(* IEC 61131-3 sources: Yaha/Documentation/Infomaterial/OSCAT/pcworx_building_100/pcworx_building_100/pcworx_building_100_module_export, 58 files *)

(* ---- building.IEC ---- *)
(*@PROPERTIES_EX@
TYPE: DATA_TYPE
LOCALE: 0
*)
(* ------------------------------------------- *)

TYPE oscat_TIMER_EVENT_DATA :
  STRUCT
	TYP          : BYTE;
	CHANNEL      : BYTE;
	DAY          : BYTE;
	START        : UDINT;
	DURATION     : TIME;
	LAND         : BYTE;
	LOR          : BYTE;
	LAST         : UDINT;
  END_STRUCT;
END_TYPE

TYPE
  oscat_TIMER_EVENT           : ARRAY [0..63]    OF oscat_TIMER_EVENT_DATA;
END_TYPE

(* ------------------------------------------- *)

TYPE
  oscat_T_AVG24         	  : ARRAY [0..47]   OF INT;

  oscat_TP4_qn                : ARRAY [0..3]    OF BOOL;

  oscat_bsa_X                 : ARRAY [0..2]    OF BYTE;
  oscat_blind_scene_array     : ARRAY [0..15]   OF oscat_bsa_X;

END_TYPE

(* ---- ACTUATOR_2P.ST ---- *)
(*@PROPERTIES_EX@
TYPE: POU
LOCALE: 0
IEC_LANGUAGE: ST
PLC_TYPE: independent
PROC_TYPE: independent
GROUP: ACTUATORS
*)
(*@KEY@:DESCRIPTION*)
version 2.1	24. jan. 2009
programmer 	hugo
tested by	oscat

this is an intelligent actuator interface for any 2point actuator like coil drive.
the 2Point actuator can only switch on/off and therefore the input must be converted to on/off cycles.
the interface can be programmed with double click on the symbol.
in addition a self_act_time and self_act_cycles ca be programmed to switch n times on/off every self_act_time to avoid a valve to freeze.
the input value must be between 0 and 255. with the setup variable sens one can specify what must be the minimum input to turn the valve on at all.
at the same time an input > 255-sens will turn the valve on at all times.
(*@KEY@:END_DESCRIPTION*)
FUNCTION_BLOCK ACTUATOR_2P

(*Group:Default*)

VAR_INPUT
	IN :	BYTE;
	TEST :	BOOL;
	ARE :	BOOL := TRUE;
	CYCLE_TIME :	TIME;
	SENS :	BYTE;
	SELF_ACT_TIME :	TIME;
	SELF_ACT_PULSE :	TIME;
	SELF_ACT_CYCLES :	INT := 1;
END_VAR

VAR_OUTPUT
	OUT :	BOOL;
	ARO :	BOOL;
END_VAR

VAR_IN_OUT
	ARX :	BOOL;
END_VAR

VAR
	timer :	AUTORUN;
	pwgen :	GEN_PULSE;
END_VAR

(*@KEY@: WORKSHEET
NAME: ACTUATOR_2P
IEC_LANGUAGE: ST
*)
(* run the autorun timer *)
timer(trun := MUL_T_AI(SELF_ACT_PULSE,2 * SELF_ACT_CYCLES), toff := SELF_ACT_TIME, Test := TEST, ARE := ARE, arx := ARX);
ARX := timer.ARX;
ARO := timer.ARO;

(* run the pulse width generator *)
IF aro THEN
	pwgen(PTL := SELF_ACT_PULSE, PTH := SELF_ACT_PULSE);
	out := pwgen.Q;
ELSIF in < sens THEN
	out := FALSE;
ELSIF BYTE_TO_USINT(in) > USINT#255 - BYTE_TO_USINT(sens) THEN
	out := TRUE;
ELSE
	pwgen.PTH := (CYCLE_TIME * BYTE_TO_TIME(BAND_B(IN,SENS))  ) / BYTE_TO_TIME(BYTE#255);
	pwgen.PTL := CYCLE_TIME - pwgen.PTH;
	pwgen();
	out := pwgen.Q;
END_IF;

(* revision history
hm	7.10.2006 		rev 1.1
	changed error pos could not reach 1 or 0 under certain conditions due to error in code.
	changed on and off in force and force_in for better usability.

hm	17.1.2007		rev 1.2
	deleted unused variable time_overflow

hm	15.9.2007		rev 1.3
	replaced time() with T_PLC_MS for compatibility and performance reasons

hm	19. 11 2007		rev 1.4
	replaced left over statement time() with tx

hm	27. 12. 2007	REV 1.5
	CHANGED CODE FOR BETTER PERFORMANCE

hm	21. oct. 2008	rev 1.6
	code optimized

hm	23. nov. 2008	rev 2.0
	new code using library modules

hm	24. jan. 2009	rev 2.1
	deleted unused var inb
*)
(*@KEY@: END_WORKSHEET *)
END_FUNCTION_BLOCK

(* ---- ACTUATOR_3P.ST ---- *)
(*@PROPERTIES_EX@
TYPE: POU
LOCALE: 0
IEC_LANGUAGE: ST
PLC_TYPE: independent
PROC_TYPE: independent
GROUP: ACTUATORS
*)
(*@KEY@:DESCRIPTION*)
version 2.0	28. jan 2010
programmer 	hugo
tested by		oscat

actuator_3P is an interface for a 3 point actuator.
a 3P actuator is a motor with 2 directions that drives a valve or flap. the position of the valve or flap is controlled by runtime of the motor foreward or backward.
the available inputs are:
IN specifies the position of the actuator, 0 = 0% and 255 = 100%.
an END_POS input is available for an end_pos switch, this switch indicates the valve or flap to be at either 0% or 100%
a TEST input can at any time start a diag cycle which turns the motor towards the 0% position, then measures the runtime to 100% and then the runtime to 0%
these runtimes are stored and used for absolute positioning of the motor during normal operation. this feature is only avaliable with an END_POS switch connected to the input.
a setup variable T_DIAG can be used to specify how often the actuator repeates this auto_diag cycle automatically.
at power on a diag cycle is perfomed automatically.
a time of 0 for T_DIAG means auto diag is never performed.

the outputs out1 and out2 are for the two directions of the motor.
a pos output indicates the simulated position of the actuator during operation.
a error output is activated when the specified max_runtime is reached by any direction during debug without an end_switch to become active.
also when the up and down direction differs by more then 10% the error output is set.

for absolute positioning accuracy the actuator has a setup variable "cal_runtime" if this is set the actuator measures the total runtime of the motors and when this
cal_runtime is exceeded it resets the actuator to 0% position and sets the output again to assure absolute accuracy.

test and calibration can be shut off by setting the appropriate values to 0.
a switch_available setup variable specifies if end_pos switches are available.
(*@KEY@:END_DESCRIPTION*)
FUNCTION_BLOCK ACTUATOR_3P

(*Group:Default*)

VAR_INPUT
	IN :	BYTE;
	TEST :	BOOL;
	ARE :	BOOL := TRUE;
	END_POS :	BOOL;
	T_RUN :	TIME := T#60s;
	T_EXT :	TIME := T#10s;
	T_CAL :	TIME := T#600s;
	T_DIAG :	TIME := T#10d;
	SWITCH_AVAIL :	BOOL;
END_VAR

VAR_OUTPUT
	OUT1 :	BOOL;
	OUT2 :	BOOL;
	POS :	BYTE;
	ERROR :	BOOL;
	STATUS :	BYTE;
END_VAR

VAR_IN_OUT
	ARX :	BOOL;
END_VAR

VAR
	tx :	TIME;
	ramp :	_RMP_NEXT;
	next_cal :	TIME;
	next_diag :	TIME;
	last :	TIME;
	start :	TIME;
	T_PLC_MS :	T_PLC_MS;
END_VAR

(*@KEY@: WORKSHEET
NAME: ACTUATOR_3P
IEC_LANGUAGE: ST
*)
(* setup *)
T_PLC_MS();
tx := UDINT_TO_TIME(T_PLC_MS.T_PLC_MS);

(* check test input *)
IF TEST THEN
	status := BYTE#103;
	start := tx;
	ARX := TRUE;
END_IF;

CASE _BYTE_TO_INT(status) OF
	0:	(* power on setup *)
		IF ARE AND NOT ARX THEN
			status := BYTE#103;
			start := tx;
			ARX := TRUE;
		END_IF;

	100:	(* normal operation *)
		(* check for auto diagnostics *)
		IF T_DIAG > T#0s AND tx > next_diag AND ARE AND NOT ARX THEN
				status := BYTE#103;
				start := tx;
				ARX := TRUE;

		(* check for auto calibration *)
		ELSIF T_CAL > T#0s AND tx > next_cal AND ARE AND NOT ARX THEN
			IF pos > BYTE#127 THEN
				OUT1 := TRUE;
				OUT2 := FALSE;
				ramp.IN := BYTE#255;
				ARX := TRUE;
			ELSE
				OUT1 := FALSE;
				OUT2 := TRUE;
				ramp.IN := BYTE#0;
				ARX := TRUE;
			END_IF;
			status := BYTE#101;
			start := tx;
		ELSE
			(* increment next_cal if not active *)
			IF NOT(OUT1 OR OUT2) THEN next_cal := next_cal + (tx-last); END_IF;
			(* set ramp generator to IN *)
			ramp.IN := IN;
		END_IF;

	101:	(* calibrate *)
		IF tx - start < T_EXT THEN
			next_cal := tx + T_CAL;
		ELSIF SWITCH_AVAIL AND END_POS THEN
			STATUS := BYTE#100;
			ARX := FALSE;
		ELSIF tx - start > T_EXT + T_RUN THEN
			ERROR := SWITCH_AVAIL;
			ARX := FALSE;
		END_IF;

	103:	(* diagnostics up*)
		(* run up for T_ext *)
		IF tx - start < T_EXT THEN
			ERROR := FALSE;
			ramp.TR := T_RUN;
			ramp.TF := T_RUN;
			OUT1 := TRUE;
			OUT2 := FALSE;
			ramp.IN := BYTE#255;
		ELSIF SWITCH_AVAIL AND END_POS THEN
			ramp.TR := tx - start;
			STATUS := BYTE#104;
		ELSIF tx - start > T_EXT + T_RUN THEN
			ERROR := SWITCH_AVAIL;
			STATUS := BYTE#104;
			start := tx;
		END_IF;

	104:	(* diagnostics dn*)
		IF tx - start < T_ext THEN
			OUT1 := FALSE;
			OUT2 := TRUE;
			ramp.IN := BYTE#0;
			next_diag := tx + T_DIAG;
		ELSIF SWITCH_AVAIL AND END_POS THEN
			ramp.TR := tx - start;
			(* check if runtimes differ by more than 10% *)
			IF DINT_TO_TIME(ABS(TIME_TO_DINT(ramp.TR) - TIME_TO_DINT(ramp.TF)) * DINT#10) > T_RUN THEN error := TRUE; END_IF;
			STATUS := BYTE#100;
			ARX := FALSE;
			next_cal := tx + T_CAL;
		ELSIF tx - start > T_EXT + T_RUN THEN
			IF SWITCH_AVAIL THEN ERROR := TRUE; END_IF;
			STATUS := BYTE#100;
			ARX := FALSE;
			next_CAL := tx + T_CAL;
		END_IF;
END_CASE;

(* internal flap simulation and output activation *)
ramp(OUT := POS);
POS := ramp.OUT;
IF STATUS = BYTE#100 THEN
	OUT1 := ramp.UP;
	OUT2 := ramp.DN;
END_IF;

(* adjust position if end switch is active *)
IF SWITCH_AVAIL AND END_POS THEN
	POS := SEL_BYTE(POS > BYTE#127, BYTE#0, BYTE#255);
	next_cal := tx + T_CAL;
END_IF;

(* set last to tx for next cycle *)
last := tx;

(* revision history

hm	19. oct 2006	rev 1.1
	added security checks for end_switch to avoid overrun of the end_switch, hans

hm	23. jan 2007	rev 1.2
	deleted unused variables force_on and force_off

hm	15. sep 2007	 rev 1.3
	replaced Time() with T_PLC_MS for compatibility and performance reasons

hm	28. jan 2010	rev 2.0
	new code and new features

*)
(*@KEY@: END_WORKSHEET *)
END_FUNCTION_BLOCK

(* ---- ACTUATOR_A.ST ---- *)
(*@PROPERTIES_EX@
TYPE: POU
LOCALE: 0
IEC_LANGUAGE: ST
PLC_TYPE: independent
PROC_TYPE: independent
GROUP: ACTUATORS
*)
(*@KEY@:DESCRIPTION*)
version 1.0 3. nov. 2008
programmer 	hugo
tested by	oscat

ACTUATOR_A drives any valve or similar with 0 - 100% analog control.
(*@KEY@:END_DESCRIPTION*)
FUNCTION_BLOCK ACTUATOR_A

(*Group:Default*)

VAR_INPUT
	I1 :	BYTE;
	IS :	BOOL;
	I2 :	BYTE;
	RV :	BOOL;
	DX :	BOOL;
	RUNTIME :	TIME;
	SELF_ACT_TIME :	TIME;
	OUT_MIN :	DWORD;
	OUT_MAX :	DWORD;
END_VAR

VAR_OUTPUT
	Y :	DWORD;
END_VAR

VAR
	timer :	CYCLE_4;
	dx_edge :	BOOL;
END_VAR

(*@KEY@: WORKSHEET
NAME: ACTUATOR_A
IEC_LANGUAGE: ST
*)
(* run the system timer, if self_act_time = t#0s then state is set to 0 *)
timer(T0 := RUNTIME, T1 := RUNTIME, T3 := SELF_ACT_TIME, sl := DX AND NOT dx_edge, sx := 0, S0 := SELF_ACT_TIME > t#0s);
dx_edge := dx;

CASE timer.STATE OF
	0: 	(* self act min value *)
		Y := OUT_MIN;
	1:	(* self_act max value *)
		Y := OUT_MAX;
	3:	(* normal operation *)
		IF rv THEN
			Y := UDINT_TO_DWORD(DWORD_TO_UDINT(OUT_MAX) - (DWORD_TO_UDINT(OUT_MAX) - DWORD_TO_UDINT(OUT_MIN)) * BYTE_TO_UDINT(SEL(IS, I1, I2)) / UDINT#255);
		ELSE
			Y := UDINT_TO_DWORD((DWORD_TO_UDINT(OUT_MAX) - DWORD_TO_UDINT(OUT_MIN)) * BYTE_TO_UDINT(SEL(IS, I1, I2)) / UDINT#255 + DWORD_TO_UDINT(OUT_MIN));
		END_IF;
END_CASE;

(*
hm 	3. nov. 2008	rev 1.0
	original version

*)
(*@KEY@: END_WORKSHEET *)
END_FUNCTION_BLOCK

(* ---- ACTUATOR_COIL.ST ---- *)
(*@PROPERTIES_EX@
TYPE: POU
LOCALE: 0
IEC_LANGUAGE: ST
PLC_TYPE: independent
PROC_TYPE: independent
GROUP: ACTUATORS
*)
(*@KEY@:DESCRIPTION*)
version 1.0	1. jun. 2008
programmer 	hugo
tested by	tobias

this is an intelligent actuator interface for any coil actuator.
the coil actuator can only switch on/off.
coil actuators like vents can get stuck if they are not u8sed for a long time and need to be autoactivated on ce in a while.
(*@KEY@:END_DESCRIPTION*)
FUNCTION_BLOCK ACTUATOR_COIL

(*Group:Default*)

VAR_INPUT
	IN :	BOOL;
	SELF_ACT_CYCLE :	TIME := T#10d;
	SELF_ACT_TIME :	TIME := T#1s;
END_VAR

VAR_OUTPUT
	OUT :	BOOL;
	STATUS :	BYTE;
END_VAR

VAR
	last :	UDINT;
	init :	BOOL;
	tx :	UDINT;
	now :	UDINT;
	T_PLC_MS :	T_PLC_MS;
END_VAR

(*@KEY@: WORKSHEET
NAME: ACTUATOR_COIL
IEC_LANGUAGE: ST
*)
(* read system time *)
T_PLC_MS();
now := T_PLC_MS.T_PLC_MS;

(* initialize for first cycle *)
IF NOT init THEN
	last := now;
	init := TRUE;
ELSIF IN THEN
	OUT := TRUE;
	STATUS := BYTE#101; (* activated by input *)
	LAST := now;
ELSE
	OUT := FALSE;
	STATUS := BYTE#100; (* disabled *)
	(* now we need to check for self activation *)
	tx := now - last;
	IF (self_act_cycle > T#0s) AND (tx >= TIME_TO_UDINT(self_act_cycle)) THEN
		OUT := TRUE;
		STATUS := BYTE#102; (* auto activation *)
		IF tx >= TIME_TO_UDINT(self_act_cycle + self_act_time) THEN
			last := now;
			OUT := FALSE;
			STATUS := BYTE#100; (* idle *)
		END_IF;
	END_IF;
END_IF;

(*
revision history:

hm		1. jun. 2008 	rev 1.0
	original version

*)
(*@KEY@: END_WORKSHEET *)
END_FUNCTION_BLOCK

(* ---- ACTUATOR_PUMP.ST ---- *)
(*@PROPERTIES_EX@
TYPE: POU
LOCALE: 0
IEC_LANGUAGE: ST
PLC_TYPE: independent
PROC_TYPE: independent
GROUP: ACTUATORS
*)
(*@KEY@:DESCRIPTION*)
version 1.4		21. oct. 2008
programmer 		oscat
tested BY		oscat

actuator_pump is a pump interface which can be controlled by an input in and an input manual.
in or manual high turns the pump output on.
a rst input is used to reset the runtime counters.
when the pump was not active for a time run_every the actuator turns on the pump automatically for min_ontime.
two setup variables min_ontime and min_offtime guarantee a minimum runtime and offtime of the pump.
the units are hours and the output type is real to prevent from overfow.
(*@KEY@:END_DESCRIPTION*)
FUNCTION_BLOCK ACTUATOR_PUMP

(*Group:Default*)

VAR_INPUT
	IN :	BOOL;
	MANUAL :	BOOL;
	RST :	BOOL := FALSE;
	MIN_ONTIME :	TIME := T#10s;
	MIN_OFFTIME :	TIME := T#10s;
	RUN_EVERY :	TIME := T#10000m;
END_VAR

VAR_OUTPUT
	PUMP :	BOOL;
	RUNTIME :	UDINT;
	CYCLES :	UDINT;
END_VAR

VAR
	tx :	TIME;
	last_change :	TIME;
	meter :	ontime;
	old_man :	BOOL;
	init :	BOOL;
	T_PLC_MS :	T_PLC_MS;
END_VAR

(*@KEY@: WORKSHEET
NAME: ACTUATOR_PUMP
IEC_LANGUAGE: ST
*)
T_PLC_MS();
tx:= UDINT_TO_TIME(T_PLC_MS.T_PLC_MS);

IF NOT init THEN
	init := TRUE;
	last_change := tx;
ELSIF rst THEN
	rst := FALSE;
	runtime := UDINT#0;
	cycles := UDINT#0;
ELSIF manual AND NOT pump AND NOT old_man THEN
	last_change := tx;
	pump := TRUE;
ELSIF NOT manual AND old_man AND pump AND NOT in THEN
	last_change := tx;
	pump := FALSE;
ELSIF in AND NOT pump AND tx - last_change >= min_offtime THEN
	last_change := tx;
	pump := TRUE;
ELSIF pump AND NOT in AND NOT manual AND tx - last_change >= min_ontime THEN
	last_change := tx;
	pump := FALSE;
ELSIF NOT pump AND (tx - last_change >= run_every) AND (run_every > T#0s) THEN
	last_change := tx;
	pump := TRUE;
END_IF;

meter(in := pump, SECONDS := runtime, CYCLES := cycles);
cycles := meter.CYCLES;
runtime := meter.SECONDS;

old_man := manual;

(*
hm	27.12.2006		rev 1.1
	fixed a failure while the pump would run for tmin after startup.

hm	15.9.2007		rev 1.2
	replaced Time() with T_PLC_MS for compatibility and performance reasons

hm	13. oct. 2008	rev 1.3
	auto activation can now be disabled when run_every = t#0s

hm	21. oct. 2008	rev 1.4
	changed to use ontime rev 2.0

*)
(*@KEY@: END_WORKSHEET *)
END_FUNCTION_BLOCK

(* ---- ACTUATOR_UD.ST ---- *)
(*@PROPERTIES_EX@
TYPE: POU
LOCALE: 0
IEC_LANGUAGE: ST
PLC_TYPE: independent
PROC_TYPE: independent
GROUP: ACTUATORS
*)
(*@KEY@:DESCRIPTION*)
version 1.3	17. oct. 2008
programmer 	hugo
tested by	tobias

out_ud is a up/dn or Right/left locked output driver.
it can be controlled by automatic inputs UD and ON as well as manual inputs for up and dn.
a security input to shut off at any time is prvided by the off input.
two time set inputs ton and toff specify a minimum on time for outputs and a minimum off time before the next output can become active.
the module assures that only one output can be active at any time.
for higher security pls make sure you use hardware locking of the outputs to prevent from defective wiring or outputs.
further security is provided b feedback inputs Yup_in and Ydn_in which are separate inputs for the output signal, if these inputs are not available
pls connect them directly to Yup and Ydn.
manual mode will override automatic mode by setting the manual input high.
a status output will be 0 for normal operation or 1 - 99 for error reporting and 101 - 199 for status reporting
The status output is ESR comptible.
(*@KEY@:END_DESCRIPTION*)
FUNCTION_BLOCK ACTUATOR_UD

(*Group:Default*)

VAR_INPUT
	UD :	BOOL;
	ON :	BOOL;
	MANUAL :	BOOL;
	UP :	BOOL;
	DN :	BOOL;
	OFF :	BOOL;
	YUP_IN :	BOOL;
	YDN_IN :	BOOL;
	TON :	TIME;
	TOFF :	TIME;
	OUT_RETURN :	BOOL;
END_VAR

VAR_OUTPUT
	YUP :	BOOL;
	YDN :	BOOL;
	STATUS :	BYTE;
END_VAR

VAR
	tx :	TIME;
	last :	TIME;
	init :	BOOL;
	T_PLC_MS :	T_PLC_MS;
END_VAR

(*@KEY@: WORKSHEET
NAME: ACTUATOR_UD
IEC_LANGUAGE: ST
*)
T_PLC_MS();
tx:= UDINT_TO_TIME(T_PLC_MS.T_PLC_MS);

IF NOT init THEN
	(* INITIALIZATION AT FIRST CALL *)
	last := tx;
	init := TRUE;
ELSIF off THEN
	(* emergency shut off detected *)
	Yup := FALSE;
	Ydn := FALSE;
	last := tx;
	status := BYTE#101;

(* WATH FOR MIN TON TIME *)
ELSIF ((Yup OR Ydn) AND tx - last < Ton) THEN RETURN;
ELSIF NOT yup AND NOT ydn AND tx - last < toff THEN	RETURN;

(* manual operation *)
ELSIF manual THEN
	status := BYTE#102;
	(* directional chage set both outs 0 first *)
	IF yup AND NOT up OR ydn AND NOT dn THEN
		ydn := FALSE;
		yup := FALSE;
		last := tx;
	(* manual up operation *)
	ELSIF UP AND NOT DN AND NOT OFF THEN
		Ydn := FALSE;
		Yup := TRUE;
		last := tx;
		status := BYTE#103;
	(* manual down operation *)
	ELSIF DN AND NOT UP AND NOT OFF THEN
		Yup := FALSE;
		Ydn := TRUE;
		last := tx;
		status := BYTE#104;
	(* maual mode but no up or down *)
	ELSE
		IF YUP OR YDN THEN LAST := tx; END_IF;
		Yup := FALSE;
		Ydn := FALSE;
	END_IF;

(* automatic operation *)
ELSE
	(* directional change set outputs low first *)
	IF yup AND NOT ud OR ydn AND UD THEN
		yup := FALSE;
		ydn := FALSE;
		last := tx;
	(* automatic up operation *)
	ELSIF Ud AND on AND NOT OFF THEN
		Ydn := FALSE;
		Yup := TRUE;
		last := tx;
		status := BYTE#111;

	(* automatic down operation *)
	ELSIF NOT UD AND on AND NOT OFF THEN
		Yup := FALSE;
		Ydn := TRUE;
		last := tx;
		status := BYTE#112;
	(* standby mode *)
	ELSE
		IF Yup OR Ydn THEN last := tx; END_IF;
		Yup := FALSE;
		Ydn := FALSE;
		status := BYTE#110;
	END_IF;
END_IF;

(* make sure Yup and Ydn are never on at the same time *)
IF Ydn AND Yup_in AND out_return THEN
	Ydn := FALSE;
	status := BYTE#1;
END_IF;
IF Yup AND Ydn_in AND out_return THEN
	Yup := FALSE;
	status := BYTE#2;
END_IF;

(* revision history
hm 22. jan 2007	rev 1.1
	added status output
	changed inputs ton, toff to config variables
	added config var out_return to enable yup_in and Ydn_in
	manual mod will override automatic mode

hm	15.9.2007	rev 1.2
	replaced Time() with T_PLC_MS for compatibility and performance reasons

hm	17. oct. 2008	rev 1.3
	deleted unnecessary initialization with 0
*)
(*@KEY@: END_WORKSHEET *)
END_FUNCTION_BLOCK

(* ---- AUTORUN.ST ---- *)
(*@PROPERTIES_EX@
TYPE: POU
LOCALE: 0
IEC_LANGUAGE: ST
PLC_TYPE: independent
PROC_TYPE: independent
GROUP: ACTUATORS
*)
(*@KEY@:DESCRIPTION*)
version 1.0	20. nov 2008
programmer 	hugo
tested by	oscat
(*@KEY@:END_DESCRIPTION*)
FUNCTION_BLOCK AUTORUN

(*Group:Default*)

VAR_INPUT
	IN :	BOOL;
	TEST :	BOOL;
	ARE :	BOOL := TRUE;
	TRUN :	TIME;
	TOFF :	TIME;
END_VAR

VAR_OUTPUT
	OUT :	BOOL;
	ARO :	BOOL;
END_VAR

VAR_IN_OUT
	ARX :	BOOL;
END_VAR

VAR
	timer :	_RMP_B;
	val :	BYTE;
END_VAR

(*@KEY@: WORKSHEET
NAME: AUTORUN
IEC_LANGUAGE: ST
*)
(* run the integrator when T_off > T#0s *)
IF TOFF > T#0s THEN
	timer(DIR:= OUT, TR := SEL(OUT, TOFF, TRUN), RMP := val);
	val := timer.RMP;
ELSE
	val := BYTE#255;
END_IF;

(* when timer = 0 or test then initiate autorun until timer reaches 255 *)
IF (NOT ARX AND ARE AND val = BYTE#0) OR TEST THEN
	val := BYTE#0;
	ARO := TRUE;
	ARX := TRUE;
ELSIF val = BYTE#255 AND ARO THEN
	ARO := FALSE;
	ARX := FALSE;
END_IF;

(* output is true when autorun ARO is true or in = TRUE *)
out := IN OR ARO;

(* revision history
hm 20. nov. 2008	rev 1.0
	original version

*)
(*@KEY@: END_WORKSHEET *)
END_FUNCTION_BLOCK

(* ---- BLIND_ACTUATOR.ST ---- *)
(*@PROPERTIES_EX@
TYPE: POU
LOCALE: 0
IEC_LANGUAGE: ST
PLC_TYPE: independent
PROC_TYPE: independent
GROUP: JALOUSIE
*)
(*@KEY@:DESCRIPTION*)
version 1.4	08. mar. 2010
programmer 	AE
tested by	AE

blind actuator drives the up and down motor of a blind. T_lockout specifies the time between up or dn becomes active.
To change direction there must be a minimum wait time to allow the motors to come to rest first.
the up and down outputs QU and QD are controlled by the inputs UP and DN.
the outputs pos and ang simulate the position of the blind pos = 0 means blind is down and pos = 255 = blind is up.
the angle 0 means vertical posisition of the slates and 255 means horizontal position of the slates.
(*@KEY@:END_DESCRIPTION*)
FUNCTION_BLOCK BLIND_ACTUATOR

(*Group:Default*)

VAR_INPUT
	UP :	BOOL;
	DN :	BOOL;
	S_IN :	BYTE;
	T_UD :	TIME := T#10s;
	T_ANGLE :	TIME := T#3s;
	T_LOCKOUT :	TIME := t#100ms;
END_VAR

VAR_OUTPUT
	POS :	BYTE;
	ANG :	BYTE;
	QU :	BOOL;
	QD :	BOOL;
	STATUS :	BYTE;
END_VAR

VAR
	position :	rmp_B;
	angle :	rmp_B;
	lock :	interlock;
END_VAR

(*@KEY@: WORKSHEET
NAME: BLIND_ACTUATOR
IEC_LANGUAGE: ST
*)
(* make sure only one motor is active at a given time *)
lock(i1 := UP, I2 := DN, TL := T_lockout);

(* ramp up or down to simulate the angle position of the blind slats *)
angle(e := lock.Q1 OR lock.Q2, UP := lock.Q1, PT := T_Angle);
position(e := lock.Q1 AND angle.high OR lock.Q2 AND angle.low, up := lock.Q1, PT := T_UD);

(* set the outputs *)
pos := position.Out;
ang := angle.Out;

(* set the outputs *)
QU := lock.Q1;
QD := lock.Q2;

(* set the status output *)
IF UP AND DN THEN
	 status := BYTE#1;			(* error up and down together are not allowed *)
ELSIF UP THEN
	status := BYTE#121;
ELSIF DN THEN
	status := BYTE#122;
ELSE
	status := S_IN;
END_IF;

(* revision history
hm	29. sep 2007	rev 1.0
	original release

hm	6. oct 2007	rev 1.1
	rearanged outputs

hm	18. oct. 2008	rev 1.2
	changed calls for rmp_B because of change in RMP_B

hm	27. jul. 2009	rev 1.3
	changes status to be 12X

ae	08. mar. 2010 rev 1.4
	at aPosition

*)
(*@KEY@: END_WORKSHEET *)
END_FUNCTION_BLOCK

(* ---- BLIND_CONTROL.ST ---- *)
(*@PROPERTIES_EX@
TYPE: POU
LOCALE: 0
IEC_LANGUAGE: ST
PLC_TYPE: independent
PROC_TYPE: independent
GROUP: JALOUSIE
*)
(*@KEY@:DESCRIPTION*)
version 1.5		8. mar 2011
programmer 		AE
tested by		AE
(*@KEY@:END_DESCRIPTION*)
FUNCTION_BLOCK BLIND_CONTROL

(*Group:Default*)

VAR_INPUT
	UP :	BOOL;
	DN :	BOOL;
	S_IN :	BYTE;
	PI :	BYTE;
	AI :	BYTE;
	T_UD :	TIME;
	T_ANGLE :	TIME;
	SENS :	BYTE := 5;
	T_LOCKOUT :	TIME := T#100ms;
END_VAR

VAR_OUTPUT
	POS :	BYTE;
	ANG :	BYTE;
	MU :	BOOL;
	MD :	BOOL;
	STATUS :	BYTE;
END_VAR

VAR
	act :	blind_actuator;
	delta :	BYTE;
	bTimeTest :	BOOL;
	iPos :	BYTE;
	iAngel :	BYTE;
END_VAR

(*@KEY@: WORKSHEET
NAME: BLIND_CONTROL
IEC_LANGUAGE: ST
*)
IF bTimeTest THEN
	PI:=iPos;
	AI:=iAngel;
	UP:=TRUE;
	DN:=TRUE;
END_IF;

(* Check Position*)
act(T_UD:=T_UD, T_ANGLE:=T_ANGLE, T_lockout := T_Lockout);

IF UP AND DN THEN
	(* automatic modus detected *)
	(* first find correct position *)
	IF _BYTE_TO_INT(act.pos) < _BYTE_TO_INT(pi) - _BYTE_TO_INT(delta) THEN
		act.UP := TRUE;
		act.DN := FALSE;
		delta := BYTE#0;
		STATUS := BYTE#121;
	ELSIF _BYTE_TO_INT(act.pos) > _BYTE_TO_INT(pi) + _BYTE_TO_INT(delta) THEN
		act.UP := FALSE;
		act.DN := TRUE;
		delta := BYTE#0;
		STATUS := BYTE#122;
	(* regulate angle *)
	ELSIF _BYTE_TO_INT(act.ang) < _BYTE_TO_INT(ai) - _BYTE_TO_INT(delta) AND T_angle > T#100ms THEN
		act.UP := TRUE;
		act.DN := FALSE;
		delta := SHR(sens,2);
		STATUS := BYTE#123;
	ELSIF _BYTE_TO_INT(act.ang) > _BYTE_TO_INT(ai) + _BYTE_TO_INT(delta) AND T_angle > T#100ms THEN
		act.UP := FALSE;
		act.DN := TRUE;
		delta := SHR(sens,2);
		STATUS := BYTE#124;
	(* correct position reached *)
	ELSE
		act.UP := FALSE;
		act.DN := FALSE;
		delta := sens;
		STATUS := S_IN;
	END_IF;
ELSE
	act.UP := UP;
	act.DN := DN;
	STATUS := S_IN;
END_IF;

(* blind control calls blind_actuator *)
act(T_UD:=T_UD, T_ANGLE:=T_ANGLE, T_lockout := T_Lockout);
pos := act.pos;
ang := act.ang;
MU := act.QU;
md := act.QD;
status := act.status;

(* revision history
hm	29. sep 2007	rev 1.0
	original release

hm	6. oct 2007	rev 1.1
	rearranged outputs
	integrated blind_actuator into blind_control

hm	16. oct 2007	rev 1.2
	ignore angle when t_angle = 0

hm 29. oct 2007	rev 1.3
	added lockout configuration time for motor direction change
	sens has a setup value of 5

hm	27. jul. 2009	rev 1.4
	changed status handling

ae	08. mar. 2010	rev 1.5
	at aPosition bevor control
	at tolerance "delta := sens/2;"

*)
(*@KEY@: END_WORKSHEET *)
END_FUNCTION_BLOCK

(* ---- BLIND_CONTROL_S.ST ---- *)
(*@PROPERTIES_EX@
TYPE: POU
LOCALE: 0
IEC_LANGUAGE: ST
PLC_TYPE: independent
PROC_TYPE: independent
GROUP: JALOUSIE
*)
(*@KEY@:DESCRIPTION*)
version 1.2	23. jan 2010
programmer 	hugo
tested by	heinz
(*@KEY@:END_DESCRIPTION*)
FUNCTION_BLOCK BLIND_CONTROL_S

(*Group:Default*)

VAR_INPUT
	UP :	BOOL;
	DN :	BOOL;
	S_IN :	BYTE := BYTE#125;
	PI :	BYTE;
	T_UP :	TIME;
	T_DN :	TIME;
	RU :	BOOL;
	RD :	BOOL;
	T_LOCKOUT :	TIME := T#100ms;
	T_EXT :	TIME;
	EXT_TRIG :	BYTE := BYTE#5;
	R_POS_TOP :	BYTE := BYTE#255;
	R_POS_BOT :	BYTE;
END_VAR

VAR_OUTPUT
	POS :	BYTE;
	MU :	BOOL;
	MD :	BOOL;
	STATUS :	BYTE;
END_VAR

VAR
	T_PLC_MS :	T_PLC_MS;
	rmp :	_RMP_NEXT;
	tx :	TIME;
	last :	TIME;
	pi_last :	BYTE;
END_VAR

(*@KEY@: WORKSHEET
NAME: BLIND_CONTROL_S
IEC_LANGUAGE: ST
*)
(* status definition
	121 = manual up				manual up operation UP = true and DN = false
	122 = manual down			manual down operation DN = true and UP = false
	123 = auto positioning		automatic mode DN = UP = TRUE
	124 = revert					revert from top or bottom
	125 = nothing					default input for S_IN
	127 = Lockout time			lockout between directional change
	128 = calibrate				calibrate after power up
	129 = extend					extend runtime at top or bottom for continuous calibration
*)

(* read system time *)
T_PLC_MS();
tx:= UDINT_TO_TIME(T_PLC_MS.T_PLC_MS);

(* check inputs and start state machine *)
IF UP  AND NOT DN THEN
	(*  manual UP *)
	rmp.IN := BYTE#255;
	STATUS := BYTE#121;
ELSIF DN AND NOT UP THEN
	(* manual DN *)
	rmp.IN := BYTE#0;
	STATUS := BYTE#122;
ELSIF NOT (UP OR DN) THEN
	(* manual standby mode *)
	rmp.IN := PI;
	STATUS := S_IN;
END_IF;

(* simulate pos output *)
rmp(E := UP OR DN, TR := T_UP, TF := T_DN, TL := T_LOCKOUT, OUT := POS);
pos := rmp.OUT;

(* state machine *)
CASE _BYTE_TO_INT(STATUS) OF
	0:		(* power up init *)
		last := tx;
		PI_last := PI XOR BYTE#255;
		STATUS := BYTE#128;		(* calibrate *)

	121: 	(* manual up *)
		MU := TRUE;
		MD := FALSE;
		IF POS >= USINT_TO_BYTE(USINT#255 - BYTE_TO_USINT(EXT_TRIG)) THEN
			(* extend cycle if top is reached *)
			POS := BYTE#255;
			last := tx;
			STATUS := BYTE#129;	(* extend *)
		END_IF;

	122:	(* manual down *)
		MD := TRUE;
		MU := FALSE;
		IF POS <= EXT_TRIG THEN
			(* extend cycle if bottom is reached *)
			POS := BYTE#0;
			last := tx;
			STATUS := BYTE#129;	(* extend *)
		END_IF;

	123:	(* auto positioning *)
		MD := rmp.DN;
		MU := rmp.UP;
		IF NOT (rmp.DN OR rmp.UP) THEN
			(* automatic position is reached *)
			IF POS <= EXT_TRIG THEN
				(* extend at bottom *)
				MD := TRUE;
				last := tx;
				STATUS := BYTE#129;	(* extend *)
			ELSIF POS >= USINT_TO_BYTE(USINT#255 - BYTE_TO_USINT(EXT_TRIG)) THEN
				(* extend at top *)
				MU := TRUE;
				last := tx;
				STATUS := BYTE#129;	(* extend *)
			ELSE
				STATUS := S_IN;
			END_IF;
		END_IF;

	124:	(* revert from top or bottom *)
		MD := rmp.DN;
		MU := rmp.UP;
		IF NOT(rmp.DN OR rmp.UP) THEN
(*		IF POS = rmp.IN THEN  *)
			PI_last := PI;
			STATUS := S_IN;
		END_IF;

	127:	(* lockout time *)
		IF (tx - last) >= T_LOCKOUT THEN
				STATUS := S_IN;
		END_IF;

	128:	(* calibration *)
		MU := TRUE;
		MD := FALSE;
		rmp.IN := BYTE#255;
		IF (tx - last) >= (T_UP +  T_EXT) THEN
			MU := FALSE;
			last := tx;
			STATUS := BYTE#127;	(* lockout *)
		END_IF;

	129: (* extend mode *)
		IF (tx - last) >= T_EXT THEN
			MU := FALSE;
			MD := FALSE;
			last := tx;
			STATUS := BYTE#127;	(* lockout *)
		END_IF;

ELSE
	MU := FALSE;
	MD := FALSE;
	IF PI <> PI_last THEN
		PI_last := PI;
		rmp.IN := PI;
		STATUS := BYTE#123;	(* auto positioning *)
	ELSIF POS = BYTE#0 AND RU THEN
		rmp.IN := R_POS_BOT;
		STATUS := BYTE#124;	(* revert *)
	ELSIF pos = BYTE#255 AND RD THEN
		rmp.IN := R_POS_TOP;
		STATUS := BYTE#124;	(* revert *)
	ELSE
		STATUS := S_IN;
	END_IF;
END_CASE;

(* revision history

hm	9. mar. 2009	rev 1.0
	original release

hf	27. jul 2009	rev 1.1
	major code changes and updates

hf	23. Jan 2010	rev 1.2
	fixed a bug during calibration
	added T_UP and T_DN

*)
(*@KEY@: END_WORKSHEET *)
END_FUNCTION_BLOCK

(* ---- BLIND_INPUT.ST ---- *)
(*@PROPERTIES_EX@
TYPE: POU
LOCALE: 0
IEC_LANGUAGE: ST
PLC_TYPE: independent
PROC_TYPE: independent
GROUP: JALOUSIE
*)
(*@KEY@:DESCRIPTION*)
version 1.7	12. nov. 2009
programmer 	hugo
tested by	oscat
(*@KEY@:END_DESCRIPTION*)
FUNCTION_BLOCK BLIND_INPUT

(*Group:Default*)

VAR_INPUT
	POS :	BYTE;
	ANG :	BYTE;
	S1 :	BOOL;
	S2 :	BOOL;
	IN :	BOOL;
	PI :	BYTE;
	AI :	BYTE;
	SINGLE_SWITCH :	BOOL;
	CLICK_EN :	BOOL := TRUE;
	CLICK_TIME :	TIME := T#500ms;
	MAX_RUNTIME :	TIME := T#60s;
	MANUAL_TIMEOUT :	TIME := T#1h;
	DEBOUNCE_TIME :	TIME := T#20ms;
	DBL_CLK1 :	BOOL := FALSE;
	DBL_POS1 :	BYTE;
	DBL_ANG1 :	BYTE;
	DBL_CLK2 :	BOOL := FALSE;
	DBL_POS2 :	BYTE := BYTE#255;
	DBL_ANG2 :	BYTE := BYTE#255;
	D1_TOGGLE :	BOOL := TRUE;
	D2_TOGGLE :	BOOL := TRUE;
	MASTER_MODE :	BOOL;
END_VAR

VAR_OUTPUT
	QU :	BOOL := TRUE;
	QD :	BOOL := TRUE;
	STATUS :	BYTE;
	PO :	BYTE := BYTE#255;
	AO :	BYTE := BYTE#255;
	D1 :	BOOL;
	D2 :	BOOL;
END_VAR

VAR
	s1e :	TOF;
	s2e :	TOF;
	s1d :	CLICK_MODE;
	s2d :	CLICK_MODE;
	dir :	BOOL;
	tx :	TIME;
	last :	TIME;
	T_PLC_MS :	T_PLC_MS;
END_VAR

(*@KEY@: WORKSHEET
NAME: BLIND_INPUT
IEC_LANGUAGE: ST
*)
(* read system Time *)
T_PLC_MS();
tx:= UDINT_TO_TIME(T_PLC_MS.T_PLC_MS);

(* inputs S1 and S2 are debounced and then decoded for multiple clicks *)
s1e(in := S1, pt := DEBOUNCE_TIME);
s2e(in := S2, pt := DEBOUNCE_TIME);
s1d(in := (s1e.Q AND NOT SINGLE_SWITCH) OR (s1e.Q AND SINGLE_SWITCH AND dir), t_long := CLICK_TIME);
s2d(in := (s2e.Q AND NOT SINGLE_SWITCH) OR (s1e.Q AND SINGLE_SWITCH AND NOT dir), t_long := CLICK_TIME);

(* if d1 and d2 are not toggle clear them to make sure they are only active for oine cycle *)
IF NOT d1_toggle THEN d1 := FALSE; END_IF;
IF NOT d2_toggle THEN d2 := FALSE; END_IF;

(* decode actions *)
IF (s1d.LONG AND s2d.LONG) OR (status = BYTE#139) THEN
   status := BYTE#139;
   IF NOT (s1d.LONG OR s2d.LONG)  THEN status := BYTE#130; END_IF;
ELSIF s1d.tp_LONG THEN
	status := BYTE#132;
ELSIF s2d.tp_LONG THEN
	status := BYTE#133;
ELSIF  s1d.SINGLE THEN
	IF click_en THEN
		(* if running then we stop otherwise start new direction *)
		IF QU XOR QD THEN
			status := BYTE#131;
		ELSE
			status := BYTE#134;
			last := tx;
			dir := NOT dir;
		END_IF;
	END_IF;
ELSIF  s2d.SINGLE THEN
	IF click_en THEN
		(* if running then we stop otherwise start new direction *)
		IF QU XOR QD THEN
			status := BYTE#131;
		ELSE
			status := BYTE#135;
			last := tx;
			dir := NOT dir;
		END_IF;
	END_IF;
ELSIF in THEN
	status := BYTE#136;
	last := tx;
ELSIF s1d.DOUBLE THEN
	IF dbl_clk1 THEN
		(* a position need to be set for a double click on S1 *)
		status := BYTE#137;
		last := tx;
	ELSE
		(* toggle the output when dbl_clk1 is not active *)
		D1 := NOT D1;
	END_IF;
ELSIF s2d.DOUBLE THEN
	IF dbl_clk2 THEN
		(* a position need to be set for a double click on S2 *)
		status := BYTE#138;
		last := tx;
	ELSE
		(* toggle the output when dbl_clk2 is not active *)
		(* in single switch mode we need to toggle d1 instead of d2 *)
		IF single_switch THEN D1 := NOT D1; ELSE D2 := NOT D2; END_IF;
	END_IF;
END_IF;

(* state machine *)
CASE _BYTE_TO_INT(status) OF
	0:		(* power up operation *)
			status := BYTE#130;

	130:	(* automatic operation standby *)
			IF NOT master_mode THEN
				PO := POS;
				AO := ANG;
			END_IF;
			QU := TRUE;
			QD := TRUE;

	131:	(* manual operation standby *)
			QU := FALSE;
			QD := FALSE;
			PO := POS;
			AO := ANG;
			(* manual mode will be ended when timeout is reached *)
			IF tx - last >= manual_timeout THEN
				status := BYTE#130;
			END_IF;

	132:	(* manual operation up *)
			QU := TRUE;
			QD := FALSE;
			PO := POS; AO := ANG;
			last := tx;
			IF NOT s1d.LONG THEN status := BYTE#131; dir := NOT dir; END_IF;

	133:	(* manual operation down *)
			QU := FALSE;
			QD := TRUE;
			PO := POS; AO := ANG;
			last := tx;
			IF NOT s2d.LONG THEN	status := BYTE#131; dir := NOT dir; END_IF;

	134:	(* manual operation single click up *)
			QU := TRUE;
			QD := FALSE;
			PO := POS; AO := ANG;
			IF tx - last >= max_runtime THEN status := BYTE#131; END_IF;

	135:	(* manual operation single click dn *)
			QU := FALSE;
			QD := TRUE;
			PO := POS; AO := ANG;
			IF tx - last >= max_runtime THEN status := BYTE#131;	END_IF;

	136:	(* forced input in = true *)
			QU := TRUE;
			QD := TRUE;
			PO := PI; AO := AI;
			IF tx-last >= max_runtime THEN status := BYTE#130; END_IF;

	137:	(* double click1 position *)
			QU := TRUE;
			QD := TRUE;
			PO := DBL_POS1;
			AO := DBL_ANG1;
			IF tx - last >= max_runtime THEN status := BYTE#131; END_IF;

	138:	(* double click2 position *)
			QU := TRUE;
			QD := TRUE;
			PO := DBL_POS2;
			AO := DBL_ANG2;
			IF tx - last >= max_runtime THEN status := BYTE#131; END_IF;

	   139:   (* manual operation standby *)
	         QU := FALSE;
	         QD := FALSE;
	         PO := POS;
	         AO := ANG;

END_CASE;

(* revision history
hm	29. sep 2007	rev 1.0
	original release

hm	6. oct 2007		rev 1.1
	renamed ps and as to po and ao

hm	30. dec 2007	rev 1.2
	added click_timeout variable and function

hm	16. jul. 2008	rev 1.3
	rewirtten code to allow for more functionality
	added single click mode with single_switch.
	added Debounce for inputs S1 and S2
	added double_click functionality

hm	26. sep. 2008	rev 1.4
	corrected an error while POS and ANG was transferred to outputs PO and AO during automatic modes

hm	22. jan 2009	rev 1.5
	added pulse mode for double click outputs
	added automatic mode for IN

hm	27. jul 2009	rev 1.6
	changed status 0 to 130

HF	12. nov. 2009	rev 1.7
	added state 139
	set defaults for QU, QD, PO

*)
(*@KEY@: END_WORKSHEET *)
END_FUNCTION_BLOCK

(* ---- BLIND_NIGHT.ST ---- *)
(*@PROPERTIES_EX@
TYPE: POU
LOCALE: 0
IEC_LANGUAGE: ST
PLC_TYPE: independent
PROC_TYPE: independent
GROUP: JALOUSIE
*)
(*@KEY@:DESCRIPTION*)
version 1.2	6 oct 2007
programmer 	hugo
tested by	tobias
(*@KEY@:END_DESCRIPTION*)
FUNCTION_BLOCK BLIND_NIGHT

(*Group:Default*)

VAR_INPUT
	UP :	BOOL;
	DN :	BOOL;
	S_IN :	BYTE;
	PI :	BYTE;
	AI :	BYTE;
	E_NIGHT :	BOOL := TRUE;
	E_DAY :	BOOL := TRUE;
	DTIN :	UDINT;
	SUNRISE :	UDINT;
	SUNSET :	UDINT;
	SUNRISE_OFFSET :	TIME;
	SUNSET_OFFSET :	TIME;
	NIGHT_POSITION :	BYTE;
	NIGHT_ANGLE :	BYTE;
END_VAR

VAR_OUTPUT
	QU :	BOOL;
	QD :	BOOL;
	STATUS :	BYTE;
	PO :	BYTE;
	AO :	BYTE;
END_VAR

VAR
	night :	BOOL;
	last_night :	UDINT;
	last_day :	UDINT;
END_VAR

(*@KEY@: WORKSHEET
NAME: BLIND_NIGHT
IEC_LANGUAGE: ST
*)
IF NOT (up AND dn) AND night THEN
	(* manual operation at night will cancel operation for one night *)
	night := FALSE;
ELSIF (DT_TO_TOD(dtin) > sunset + TIME_TO_UDINT(sunset_offset)) AND (last_night < DT_TO_DATE(dtin)) AND NOT night AND e_night THEN
	(* enable night *)
	night := TRUE;
	last_night := DT_TO_DATE(dtin);
ELSIF (DT_TO_TOD(dtin) > sunrise + TIME_TO_UDINT(sunrise_offset)) AND (last_day < DT_TO_DATE(dtin)) AND night AND e_day AND (last_night < DT_TO_DATE(dtin)) THEN
	(* disable night *)
	night := FALSE;
	last_day := DT_TO_DATE(dtin);
END_IF;

(* shade at night only in auto mode and enable = true *)
IF UP AND DN AND night THEN
	status := BYTE#141;
	po := night_position;
	ao := night_angle;
ELSE
	QU := UP;
	QD := DN;
	po := pi;
	ao := ai;
	status := s_in;
END_IF;

(* revision history
hm	29. sep 2007	rev 1.0
	original version

hm	5. oct 2007		rev 1.1
	added enable input

hm	6. oct 2007		rev 1.2
	added pos and angle inputs and outputs
	night position and angle can now be configured
	any manual operation at night will cancel night operation

*)
(*@KEY@: END_WORKSHEET *)
END_FUNCTION_BLOCK

(* ---- BLIND_SCENE.ST ---- *)
(*@PROPERTIES_EX@
TYPE: POU
LOCALE: 0
IEC_LANGUAGE: ST
PLC_TYPE: independent
PROC_TYPE: independent
GROUP: JALOUSIE
*)
(*@KEY@:DESCRIPTION*)
version 1.1	29. jan 2008
programmer 	hugo
tested by	tobias
(*@KEY@:END_DESCRIPTION*)
FUNCTION_BLOCK BLIND_SCENE

(*Group:Default*)

VAR_INPUT
	UP :	BOOL;
	DN :	BOOL;
	S_IN :	BYTE;
	PI :	BYTE;
	AI :	BYTE;
	ENABLE :	BOOL;
	SWRITE :	BOOL;
	SCENE :	BYTE;
END_VAR

VAR_OUTPUT
	QU :	BOOL;
	QD :	BOOL;
	STATUS :	BYTE;
	PO :	BYTE;
	AO :	BYTE;
END_VAR

VAR
	x :	INT;
END_VAR

VAR RETAIN
	sx :	oscat_blind_scene_array;
END_VAR

(*@KEY@: WORKSHEET
NAME: BLIND_SCENE
IEC_LANGUAGE: ST
*)
(* delete all bits except the lower 4 of scene *)
x := _BYTE_TO_INT(scene AND BYTE#2#0000_1111);

IF enable AND (sx[x][2] > BYTE#0) AND UP AND DN THEN
	po := sx[x][0];
	ao := sx[x][1];
	status := INT_TO_BYTE(160 + x);  (* Status number is 160 to 175 for the 16 scenes *)
	QU := TRUE;
	QD := TRUE;
ELSE
	QU := UP;
	QD := DN;
	status := S_IN;
	po := pi;
	ao := ai;
END_IF;

(* write scene if necessary *)
IF swrite THEN
	status := BYTE#176;		(* write scene *)
	sx[x][0] := pi;
	sx[x][1] := ai;
	IF enable THEN sx[x][2] := BYTE#1; ELSE sx[x][2] := BYTE#0; END_IF; (* if sx[x][2] = 0 the scene is disabled *)
END_IF;

(* revision history
hm	24. oct 2007	rev 1.0
	original release

*)
(*@KEY@: END_WORKSHEET *)
END_FUNCTION_BLOCK

(* ---- BLIND_SECURITY.ST ---- *)
(*@PROPERTIES_EX@
TYPE: POU
LOCALE: 0
IEC_LANGUAGE: ST
PLC_TYPE: independent
PROC_TYPE: independent
GROUP: JALOUSIE
*)
(*@KEY@:DESCRIPTION*)
version 1.2	12. feb 2008
programmer 	hugo
tested by	tobias
(*@KEY@:END_DESCRIPTION*)
FUNCTION_BLOCK BLIND_SECURITY

(*Group:Default*)

VAR_INPUT
	UP :	BOOL;
	DN :	BOOL;
	S_IN :	BYTE;
	PI :	BYTE;
	AI :	BYTE;
	FIRE :	BOOL;
	WIND :	BOOL;
	ALARM :	BOOL;
	DOOR :	BOOL;
	RAIN :	BOOL;
	ALARM_UP :	BOOL := TRUE;
	WIND_UP :	BOOL := TRUE;
	RAIN_UP :	BOOL := TRUE;
END_VAR

VAR_OUTPUT
	QU :	BOOL;
	QD :	BOOL;
	STATUS :	BYTE;
	PO :	BYTE;
	AO :	BYTE;
END_VAR

(*@KEY@: WORKSHEET
NAME: BLIND_SECURITY
IEC_LANGUAGE: ST
*)
IF Fire THEN
	QU := TRUE;
	QD := FALSE;
	status := BYTE#111;
ELSIF Wind THEN
	QU := Wind_up;
	QD := NOT wind_up;
	status := BYTE#112;
ELSIF alarm THEN
	QU := Alarm_up;
	QD := NOT Alarm_up;
	status := BYTE#113;
ELSIF Door THEN
	QU := TRUE;
	QD := FALSE;
	status := BYTE#114;
ELSIF Rain AND NOT (up XOR dn) THEN
	QU := rain_up;
	QD := NOT rain_up;
	status := BYTE#115;
ELSE
	QU := UP;
	QD := DN;
	status := S_IN;
	po := pi;
	ao := ai;
END_IF;

(* revision history
hm	29. sep 2007	rev 1.0
	original release

hm	6. oct 2007		rev 1.1
	added pos and angle inputs and outputs
	manual will override rain position
	alarm position can now be configured

hm		12. feb. 2008	rev 1.2
	added config variables rain_up and wind_up
	position for rain and wind is now configurable
*)
(*@KEY@: END_WORKSHEET *)
END_FUNCTION_BLOCK

(* ---- BLIND_SET.ST ---- *)
(*@PROPERTIES_EX@
TYPE: POU
LOCALE: 0
IEC_LANGUAGE: ST
PLC_TYPE: independent
PROC_TYPE: independent
GROUP: JALOUSIE
*)
(*@KEY@:DESCRIPTION*)
version 1.0	27. jul 2009
programmer 	hugo
tested by	oscat

BLIND_SET can be used to force a definite position and angle.
blind_set can be placed close to blind_control for high priority while blind_input must be always at the beginning of the chain with low priority.
(*@KEY@:END_DESCRIPTION*)
FUNCTION_BLOCK BLIND_SET

(*Group:Default*)

VAR_INPUT
	UP :	BOOL;
	DN :	BOOL;
	S_IN :	BYTE;
	PI :	BYTE;
	AI :	BYTE;
	IN :	BOOL;
	PX :	BYTE;
	AX :	BYTE;
	OVERRIDE_MANUAL :	BOOL;
	RESTORE_POSITION :	BOOL;
	RESTORE_TIME :	TIME := T#60s;
END_VAR

VAR_OUTPUT
	QU :	BOOL;
	QD :	BOOL;
	STATUS :	BYTE;
	PO :	BYTE;
	AO :	BYTE;
END_VAR

VAR
	T_PLC_MS :	T_PLC_MS;
	tx :	TIME;
	ps :	BYTE;
	as :	BYTE;
	last :	TIME;
END_VAR

(*@KEY@: WORKSHEET
NAME: BLIND_SET
IEC_LANGUAGE: ST
*)
(* read system Time *)
T_PLC_MS();
tx:= UDINT_TO_TIME(T_PLC_MS.T_PLC_MS);

(* check inputs *)
IF IN THEN
	IF override_manual OR (UP AND DN) THEN
		status := 178;
	END_IF;
END_IF;

(* state machine *)
CASE STATUS OF
	0: (* power on state *)
		status := S_IN;

	178: (* force values from PX and AX *)
		PO := PX;
		AO := AX;
		QU := TRUE;
		QD := TRUE;
		(* check for end of forced position *)
		IF NOT in THEN
			STATUS := SEL(RESTORE_POSITION, S_IN, 179);
			last := tx;
		END_IF;

	179: (* restore previous position *)
		PO := ps;
		AO := as;
		IF ((PO = PI) AND (AO = AI))  OR tx - last >= RESTORE_TIME THEN
			status := S_IN;
		END_IF;

ELSE
	(* no operation transfer inputs to outputs *)
	PO := PI;
	ps := PI;
	AO := AI;
	as := AI;
	STATUS := S_IN;
	QU := UP;
	QD := DN;
END_CASE;

(* revision history
hm	27. jul 2009	rev 1.0
	original release

*)
(*@KEY@: END_WORKSHEET *)
END_FUNCTION_BLOCK

(* ---- BLIND_SHADE.ST ---- *)
(*@PROPERTIES_EX@
TYPE: POU
LOCALE: 0
IEC_LANGUAGE: ST
PLC_TYPE: independent
PROC_TYPE: independent
GROUP: JALOUSIE
*)
(*@KEY@:DESCRIPTION*)
version 1.4	13. mar. 2009
programmer 	hugo
tested by	tobias
(*@KEY@:END_DESCRIPTION*)
FUNCTION_BLOCK BLIND_SHADE

(*Group:Default*)

VAR_INPUT
	UP :	BOOL;
	DN :	BOOL;
	S_IN :	BYTE;
	PI :	BYTE;
	AI :	BYTE;
	ENABLE :	BOOL;
	SUN :	BOOL;
	SUNRISE_OFFSET :	TIME := T#1h;
	SUNSET_PRESET :	TIME := T#1h;
	DIRECTION :	REAL := 180.0;
	ANGLE_OFFSET :	REAL := 80.0;
	SLAT_WIDTH :	REAL := 80.0;
	SLAT_SPACING :	REAL := 60.0;
	SHADE_DELAY :	TIME := T#60s;
	SHADE_POS :	BYTE;
END_VAR

VAR_OUTPUT
	QU :	BOOL;
	QD :	BOOL;
	STATUS :	BYTE;
	PO :	BYTE;
	AO :	BYTE;
END_VAR

VAR_IN_OUT
	CX :	oscat_CALENDAR;
END_VAR

VAR
	angle :	REAL;
	sun_delay :	TOF;
END_VAR

(*@KEY@: WORKSHEET
NAME: BLIND_SHADE
IEC_LANGUAGE: ST
*)
(* the input sun is sent through tof which will delay the shade for the time shade_delay *)
sun_delay(IN := sun, PT := shade_delay);

IF UP AND DN AND enable AND sun_delay.Q AND cx.SUN_HOR > direction - angle_offset AND cx.SUN_HOR < direction + angle_offset AND
	DT_TO_TOD(cx.UTC) > cx.SUN_RISE + TIME_TO_UDINT(sunrise_offset) AND DT_TO_TOD(cx.UTC) < cx.SUN_SET - TIME_TO_UDINT(sunset_preset) THEN
	status := BYTE#151;
	QU := UP;
	QD := DN;
	(* position is predefined *)
	po := shade_pos;
	(* shading is active now calculate the slat angle *)
	(* calculate the max angle for the blind *)
	angle := DEG(ATAN(slat_spacing / slat_width));
	(* check if sun angle is between 0 and max angle *)
	IF cx.SUN_VER > 0.0 AND cx.SUN_VER < angle THEN
		angle := cx.SUN_VER + DEG(ACOS(COS(RAD(cx.SUN_VER))*slat_spacing / Slat_width));
		ao := INT_TO_BYTE(LIMIT(0,UDINT_TO_INT(TRUNC_UDINT(angle * 2.833333333)), 255));
	ELSE
		ao := BYTE#255;
	END_IF;
ELSE
	QU := UP;
	QD := DN;
	po := pi;
	ao := ai;
	status := S_IN;
END_IF;

(* revision history
hm	15 oct. 2007	rev 1.0
	original version

hm	19. oct 2007	rev 1.1
	manual mode was not detected because outputs were checked and not inputs UP and DN

hm	24. nov 2007	rev 1.2
	added shade_delay to avoid constant up and down if sun is out parcially

hm	8. feb 2009	rev 1.3
	added shading position shade_pos to be configured
	changed inputs to utilize calendar data structure

hm	13. mar. 2009	rev 1.4
	improved code

*)

(*@KEY@: END_WORKSHEET *)
END_FUNCTION_BLOCK

(* ---- BLIND_SHADE_S.ST ---- *)
(*@PROPERTIES_EX@
TYPE: POU
LOCALE: 0
IEC_LANGUAGE: ST
PLC_TYPE: independent
PROC_TYPE: independent
GROUP: JALOUSIE
*)
(*@KEY@:DESCRIPTION*)
version 1.0	12. nov. 2009
programmer 	heinz
tested by	oscat
(*@KEY@:END_DESCRIPTION*)
FUNCTION_BLOCK BLIND_SHADE_S

(*Group:Default*)

VAR_INPUT
	UP :	BOOL;
	DN :	BOOL;
	S_IN :	BYTE;
	PI :	BYTE;
	ENABLE :	BOOL;
	SUN :	BOOL;
	HORZ1 :	REAL := 100.0;
	HORZ2 :	REAL := 260.0;
	VERT :	REAL := 90.0;
	ALERT :	BOOL;
	SUNRISE_OFFSET :	TIME := T#1h;
	SUNSET_PRESET :	TIME := T#1h;
	SHADE_DELAY :	TIME := T#60s;
	SHADE_POS :	BYTE;
	QU :	BOOL;
	QD :	BOOL;
	STATUS :	BYTE;
	PO :	BYTE;
END_VAR

VAR_IN_OUT
	CX :	oscat_CALENDAR;
END_VAR

(*@KEY@: WORKSHEET
NAME: BLIND_SHADE_S
IEC_LANGUAGE: ST
*)
(* status definition
   151 = shadow               move shutter down for shadowing
   152 = alert                  move shutter up by setting QU:=TRUE when door is open.
*)

(* the input sun is sent through tof which will delay the shade for the time shade_delay *)
sun_delay(IN := sun, PT := shade_delay);

IF ALERT THEN
   QU := TRUE;
   QD := FALSE;
   STATUS := BYTE#152;
ELSIF UP AND DN AND ENABLE AND sun_delay.Q
AND (CX.SUN_HOR > HORZ1) AND (CX.SUN_HOR < HORZ2)
AND (CX.SUN_VER < VERT)
AND (DT_TO_TOD(CX.UTC) > CX.SUN_RISE + sunrise_offset) AND (DT_TO_TOD(CX.UTC) < CX.SUN_SET - sunset_preset) THEN
   QU := UP;
   QD := DN;
   STATUS := BYTE#151;
   (* Calculate Position, must be shade_pos or less *)
   PO := MIN(PI, shade_pos);
ELSE
   QU := UP;
   QD := DN;
   PO := PI;
   STATUS := S_IN;
END_IF;

(* revision history
hf	12 nov. 2009	rev 1.0
	original version

*)
(*@KEY@: END_WORKSHEET *)
END_FUNCTION_BLOCK

(* ---- BOILER.ST ---- *)
(*@PROPERTIES_EX@
TYPE: POU
LOCALE: 0
IEC_LANGUAGE: ST
PLC_TYPE: independent
PROC_TYPE: independent
GROUP: HLK
*)
(*@KEY@:DESCRIPTION*)
version 1.2	13. mar. 2009
programmer 	hugo
tested by	oscat

this function block controls a hot water boiler. The Boiler can be equipped with two temperature sensors on top and bottom of the tank, T_LOWER_ENABLE must be set to True in this case.
alternatively can BOILER be configured for one (TOP) temperature sensor only (T_LOWER_ENABLE set to False).
A Pressure sensor is used to detect fresh water pressure and disable all heating if there is no water pressure. This input is dset to True by default, so if it is not used it can simply be left open.
A enable input enables the hot water heating while it is set to True. alternatively can a Ture on Req_1 or Req_2 start the heating to predefined temperatures during setup.
A low to high edge on the boost input will start heating imediately until T_upper_max is reached, it can be used to generate extra hot water when needed.
(*@KEY@:END_DESCRIPTION*)
FUNCTION_BLOCK BOILER

(*Group:Default*)

VAR_INPUT
	T_UPPER :	REAL;
	T_LOWER :	REAL;
	PRESSURE :	BOOL := TRUE;
	ENABLE :	BOOL := TRUE;
	REQ_1 :	BOOL;
	REQ_2 :	BOOL;
	BOOST :	BOOL;
	T_UPPER_MIN :	REAL := REAL#50.0;
	T_UPPER_MAX :	REAL := REAL#60.0;
	T_LOWER_ENABLE :	BOOL;
	T_LOWER_MAX :	REAL := REAL#60.0;
	T_REQUEST_1 :	REAL := REAL#70.0;
	T_REQUEST_2 :	REAL := REAL#50.0;
	T_REQUEST_HYS :	REAL := REAL#5.0;
	T_PROTECT_HIGH :	REAL := REAL#80.0;
	T_PROTECT_LOW :	REAL := REAL#10.0;
END_VAR

VAR_OUTPUT
	HEAT :	BOOL;
	ERROR :	BOOL;
	STATUS :	BYTE;
END_VAR

VAR
	edge :	BOOL;
	boost_mode :	BOOL;
	flag_0 :	BOOL;
	flag_1 :	BOOL;
	flag_2 :	BOOL;
END_VAR

(*@KEY@: WORKSHEET
NAME: BOILER
IEC_LANGUAGE: ST
*)
(* read sensors and check for valid data *)
IF t_upper > t_protect_high THEN
	status := BYTE#1;
	heat := FALSE;
	error := TRUE;
ELSIF t_upper < t_protect_low THEN
	status := BYTE#2;
	heat := TRUE;
	error := TRUE;
ELSIF t_lower > T_protect_high AND t_lower_enable THEN
	status := BYTE#3;
	heat := FALSE;
	error := TRUE;
ELSIF t_lower < t_protect_low AND t_lower_enable THEN
	status := BYTE#4;
	heat := TRUE;
	error := TRUE;
ELSIF NOT pressure THEN
	status := BYTE#5;
	heat := FALSE;
	error := TRUE;
ELSIF req_1 OR req_2 OR enable OR boost THEN
	error := FALSE;

	(* determine if heat needs to be turned on *)
	IF boost AND NOT edge AND t_upper < t_upper_max THEN
		status := BYTE#101;
		heat := TRUE;
		boost_mode := TRUE;
	ELSIF enable AND t_upper < T_upper_min THEN
		status := BYTE#102;
		heat := TRUE;
	ELSIF req_1 AND t_upper < T_request_1 THEN
		status := BYTE#103;
		heat := TRUE;
	ELSIF req_2 AND t_upper < t_request_2 THEN
		status := BYTE#104;
		heat := TRUE;
	END_IF;

	(* determine the shut off temperature *)
	IF heat THEN
		IF (enable OR boost_mode) THEN
			flag_0 := TRUE;
			IF T_lower_enable AND T_lower > T_lower_max THEN
				flag_0 := FALSE;
				boost_mode := FALSE;
			ELSIF NOT T_lower_enable AND T_upper > T_upper_max THEN
				flag_0 := FALSE;
				boost_mode := FALSE;
			END_IF;
		ELSE
			flag_0 := FALSE;
		END_IF;
		flag_1 := (req_1 AND T_upper > T_request_1 + T_request_hys) AND req_1;
		flag_2 := (req_2 AND T_upper > T_request_2 + T_request_hys) AND req_2;

		(* shut off heat if no longer needed *)
		heat := flag_0 OR flag_1 OR flag_2;
		IF heat = FALSE THEN status := BYTE#100; END_IF;
	END_IF;
ELSE
	status := BYTE#100;
	heat := FALSE;
	error := FALSE;
END_IF;
edge := boost;

(* revision history
hm	27. feb. 2007	rev 1.0
	original version

hm	16. oct. 2008	rev 1.1
	improved performance

hm	13. mar. 2009	rev 1.2
	real constants updated to new systax using dot

*)
(*@KEY@: END_WORKSHEET *)
END_FUNCTION_BLOCK

(* ---- BURNER.ST ---- *)
(*@PROPERTIES_EX@
TYPE: POU
LOCALE: 0
IEC_LANGUAGE: ST
PLC_TYPE: independent
PROC_TYPE: independent
GROUP: HLK
*)
(*@KEY@:DESCRIPTION*)
version 1.5	15 sep 2007
programmer 	oscat
tested by	oscat

burner ist eine Oel-Brenner_steuerung fuer nichtmodulierende Oelbrenner
die steuerung kann ueber setup werte programmiert werden und entsprechenden brennern angepasst werden.
die vorheizzeit ist die zeit die eine oelvorwaermung aufgeheizt wird bevor der motor gestartet wird.
der eingang oil_temp gibt an ob die oil_temp erreicht wurde, er ist default auf true und kann auch offen gelassen werden.
die vorbelueftungszeit ist die zeit die der luefter laeuft bevor die oelzufuhr freigegeben wird.
die vorzuendzeit iust diejenige zeit die die zuendung vor offnen des oelventiel gestartet wird.
nachzuendzeit ist die zeit die nach entzuendung der flamme noch gezuendet wird.
die sicherheitszeit ist die zeit nach der die oelzufuhr gesperrt wird wenn keine flamme entsteht.
nach ablauf der sicherheitszeit wird ein fehler flag gesetzt und kann erst nach der sperrzeit wieder durch einen reset geloescht werden.
waehrend der sperrzeit ist keine weitere zuendung oder einschalten moeglich.
das flag mehrfachzuendung gibt an ob eine erloschene flamme in betrieb automatisch wieder gezuendet werden soll.
der flammwaechster liegt auf eingang flamme, ein uebertemperaturschutz auf dem eingang over_temp
der betriebsstundenzaehler gibt die brennerstunden in stunden als real ausgabewer an.
der ausgang motor steuert den luefter / pumpenmotor, oil_ventil schaltet das oil ventil und zuendung schaltet die zuendung ein.

if output fail > 0 an error happened and the output has an error code:
0 :	no error
1 :	pre heating time expired and oil temp input is not true
2 :	flame monitor is active during preheating time
3 :	flame monitor active during pre_ventilation_time
4 :	no ignoition during safety time
5 :	no flame during operation
9 :	overtemp input is true
(*@KEY@:END_DESCRIPTION*)
FUNCTION_BLOCK BURNER

(*Group:Default*)

VAR_INPUT
	IN :	BOOL;
	STAGE2 :	BOOL;
	OVER_TEMP :	BOOL;
	OIL_TEMP :	BOOL := TRUE;
	FLAME :	BOOL;
	RST :	BOOL;
	RST_TIMER :	BOOL;
	PRE_HEAT_TIME :	TIME := t#5s;
	PRE_VENT_TIME :	TIME := t#15s;
	PRE_IGNITE_TIME :	TIME := t#5s;
	POST_IGNITE_TIME :	TIME := t#25s;
	STAGE2_DELAY :	TIME := t#10s;
	SAFETY_TIME :	TIME := t#5s;
	LOCKOUT_TIME :	TIME := t#10s;
	MULTIPLE_IGNITION :	BOOL := TRUE;
	KW1 :	REAL;
	KW2 :	REAL;
END_VAR

VAR_OUTPUT
	MOTOR :	BOOL;
	COIL1 :	BOOL;
	COIL2 :	BOOL;
	PRE_HEAT :	BOOL;
	IGNITE :	BOOL;
	KWH :	REAL;
	STATUS :	BYTE;
	FAIL :	BOOL;
END_VAR

VAR_IN_OUT
	RUNTIME1 :	UDINT;
	RUNTIME2 :	UDINT;
	CYCLES :	UDINT;
END_VAR

VAR
	state :	INT;
	last :	TIME;
	tx :	TIME;
	last_change :	TIME;
	timer1 :	ONTIME;
	timer2 :	ONTIME;
	oil_temp_last :	BOOL;
	cycles2 :	UDINT;
	T_PLC_MS :	T_PLC_MS;
END_VAR

(*@KEY@: WORKSHEET
NAME: BURNER
IEC_LANGUAGE: ST
*)
(* read system time *)
T_PLC_MS();
tx:= UDINT_TO_TIME(T_PLC_MS.T_PLC_MS);

(* check rst input and overtemp *)
IF rst OR over_temp OR state = 0 THEN
	IF status > BYTE#0 AND tx - last_change >= lockout_time AND rst THEN
		status := BYTE#110;
		fail := FALSE;
		state := 1;
	ELSE
		(* normaler reset *)
		motor := FALSE;
		coil1 := FALSE;
		coil2 := FALSE;
		ignite := FALSE;
		pre_heat := FALSE;
		IF over_temp THEN
			status := BYTE#9;
			fail := TRUE;
		END_IF;
		last_change := tx;
		last := tx;
		state := 1;
	END_IF;
END_IF;

(* check for timer rst and rst timer if true *)
IF rst_timer THEN
	runtime1 := UDINT#0;
	runtime2 := UDINT#0;
	cycles := UDINT#0;
	cycles2 := UDINT#0;
END_IF;

(* quit here if an error is present *)
IF (status > BYTE#0 AND status < BYTE#100) OR rst THEN RETURN; END_IF;

(* start sequence *)
CASE state OF

1:	(* in signal starts oil pre heating *)
	IF in AND flame THEN
		state := 7;
		pre_heat := FALSE;
		status := BYTE#2;
		last_change := tx;
	ELSIF in THEN
		pre_heat := TRUE;
		state := 2;
		last_change := tx;
	END_IF;

2:	(* after pre_heating time start motor *)
	IF (tx- last_change >= pre_heat_time AND oil_temp) OR (oil_temp AND NOT oil_temp_last) THEN
		motor := TRUE;
		state := 3;
		last_change := tx;
	(* pre_heat_time ist abgelaufen und oil_temp ist nicht aktiv *)
	ELSIF tx - last_change >= pre_heat_time AND NOT oil_temp THEN
		state := 7;
		pre_heat := FALSE;
		status := BYTE#1;
		last_change := tx;
	(* flame monitor cannot be active at this time *)
	ELSIF flame THEN
		state := 7;
		pre_heat := FALSE;
		status := BYTE#2;
		last_change := tx;
	END_IF;

3:	(* abwarten bis zündung eingeschaltet werden kann *)
	IF tx - last_change >= pre_vent_time - pre_ignite_time THEN
		ignite := TRUE;
		state := 4;
		last_change := tx;
	(* flame monitor cannot be active at this time *)
	ELSIF flame THEN
		state := 7;
		pre_heat := FALSE;
		motor := FALSE;
		status := BYTE#3;
		last_change := tx;
	END_IF;

4:	(* warten bis oelzufuhr geoeffnet werden darf *)
	IF tx - last_change >= pre_ignite_time THEN
		coil1 := TRUE;
		state := 5;
		last_change := tx;
	END_IF;

5:	(* warten auf flammwaechter und falls noetig abschalten *)
	IF tx - last_change >= safety_time OR flame THEN
		IF NOT flame THEN
			(* notabschaltung da flammwaechster nicht angesprochen hat *)
			state := 7;
			motor := FALSE;
			coil1 := FALSE;
			pre_heat := FALSE;
			ignite := FALSE;
			status := BYTE#4;
			last_change := tx;
		ELSE
			state := 6;
			last_change := tx;
		END_IF;
	END_IF;

6:	(* brenner läuft, flammueberwachung und nach ablauf der nachigniteszeit ignite abschalten *)
	IF NOT flame AND NOT multiple_ignition THEN
		(* notabschaltung da flammwaechster keine flamme meldet *)
		state := 7;
		motor := FALSE;
		coil1 := FALSE;
		coil2 := FALSE;
		pre_heat := FALSE;
		ignite := FALSE;
		status := BYTE#5;
		last_change := tx;
	ELSIF NOT flame AND multiple_ignition THEN
		ignite := TRUE;
		state := 5;
		coil2 := FALSE;
		last_change := tx;
	ELSE
		IF tx - last_change >= post_ignite_time THEN
			(* post_ignite_time abgelaufen, ignite abschalten *)
			ignite := FALSE;
		END_IF;
		IF tx - last_change >= stage2_delay AND stage2 THEN
			coil2 := TRUE;
		ELSE
			coil2 := FALSE;
		END_IF;
	END_IF;
END_CASE;

(* abschaltung wenn kein eingangssignal *)
IF NOT in THEN
	state := 1;
	motor := FALSE;
	coil1 := FALSE;
	coil2 := FALSE;
	ignite := FALSE;
	pre_heat := FALSE;
	last_change := tx;
END_IF;

(* runtimezähler *)
timer1(in := flame AND in AND motor AND coil1 AND NOT coil2, SECONDS := runtime1, CYCLES := cycles);
cycles := timer1.CYCLES;
runtime1 := timer1.SECONDS;

timer2(in := flame AND in AND motor AND coil1 AND coil2, SECONDS := runtime2, CYCLES := cycles2);
cycles2 := timer2.CYCLES;
runtime2 := timer2.SECONDS;

KWH := UDINT_TO_REAL(runtime1) * KW1 / 3600.0 + UDINT_TO_REAL(runtime2) * KW2 / 3600.0;

(* zeit fuer naechsten aufruf merken *)
last := tx;

(* set fail output IF ERROR and Status  if normal operation *)

IF status > BYTE#0 AND status < BYTE#100 THEN
	fail := TRUE;
ELSE
	fail := FALSE;
	IF NOT in THEN
		status := BYTE#110;
	ELSIF flame AND in AND motor AND coil2 AND coil1 THEN
		status := BYTE#113;
	ELSIF flame AND in AND motor AND coil1 THEN
		status := BYTE#112;
	ELSE
		status := BYTE#111;
	END_IF;
END_IF;

(*
31.12.2006	hm		rev 1.1
	added pre_heat timing and output
	flame monitor before ignition will generate error on status output
	added output for KWh

31.12.2006	hm		rev 1.2
	added oil_temp_input

31.12.2006	hm		rev 1.3
	changed status output to be byte instead of bool

22.1.2007		hm		rev 1.4
	renamed fail output to status
	added output cycles
	corrected an error while pre_heat would be on when an error was present
	added coil2 output and stage2 input

15.9.2007		hm		rev 1.5
	replaced Time() with T_PLC_MS for compatibility and performance reasons

hm	21. oct. 2008	rev 1.6
	changed code to use new ontime rev 2.0
*)
(*@KEY@: END_WORKSHEET *)
END_FUNCTION_BLOCK

(* ---- CLICK.ST ---- *)
(*@PROPERTIES_EX@
TYPE: POU
LOCALE: 0
IEC_LANGUAGE: ST
PLC_TYPE: independent
PROC_TYPE: independent
GROUP: ELECTRICAL
*)
(*@KEY@:DESCRIPTION*)
version 2.0	28. dec. 2008
programmer 	oscat
tested by	oscat

click checks an input for single, double or tripple click and sets the corresponding output single, doulbe or triple for the time the input stays high at the last click.
the maximum high and low time for a click can be configured with setup variables.
the input configures itself to be high or low active depending on which state the input stays longer than t_reconfig.
(*@KEY@:END_DESCRIPTION*)
FUNCTION_BLOCK CLICK

(*Group:Default*)

VAR_INPUT
	IN :	BOOL;
	T_DEBOUNCE :	TIME := T#10ms;
	T_SHORT :	TIME := T#200ms;
	T_PAUSE :	TIME := T#500ms;
	T_RECONFIG :	TIME := T#1m;
END_VAR

VAR_OUTPUT
	Q :	BOOL;
	SINGLE :	BOOL;
	DOUBLE :	BOOL;
	TRIPLE :	BOOL;
	STATUS :	BYTE;
END_VAR

VAR
	s_in :	SW_RECONFIG;
	tx :	TIME;
	state :	INT;
	last :	TIME;
	T_PLC_MS :	T_PLC_MS;
END_VAR

(*@KEY@: WORKSHEET
NAME: CLICK
IEC_LANGUAGE: ST
*)
(* reconfiguration and debounce circuitry *)
s_in(in := in, TD := T_debounce, TR := T_reconfig);

(* read system time *)
T_PLC_MS();
tx:= UDINT_TO_TIME(T_PLC_MS.T_PLC_MS);

(* count the mumber of clicks *)
IF s_in.Q XOR Q THEN
	last := tx;
	IF s_in.Q THEN state := state + 1; END_IF;
END_IF;
Q := s_in.Q;

(* set outputs *)
IF state > 0 THEN
	IF (Q AND tx - last > t_short) OR (NOT Q AND tx - last > t_pause) THEN
		CASE state OF
			1:	single := TRUE;
				status := BYTE#111;
			2:	double := TRUE;
				status := BYTE#112;
			3:	triple := TRUE;
				status := BYTE#113;
		END_CASE;
		state := 0;
	END_IF;
ELSIF NOT q THEN
	single := FALSE;
	double := FALSE;
	triple := FALSE;
	status := BYTE#110;
	last := tx;
	state := 0;
END_IF;

(* revision history

15 Feb 2007	rev 1.0	hm
	created original version

18.5.2007	rev 1.1 hm
	corrected an error while execution would stop after t_reconfig elapsed.

15.9.2007	rev 1.2 hm
	replaced Time() with T_PLC_MS for compatibility and performance reasons

28. dec. 2008	rev 2.0
	rewritten using modular approach

*)
(*@KEY@: END_WORKSHEET *)
END_FUNCTION_BLOCK

(* ---- CLICK_MODE.ST ---- *)
(*@PROPERTIES_EX@
TYPE: POU
LOCALE: 0
IEC_LANGUAGE: ST
PLC_TYPE: independent
PROC_TYPE: independent
GROUP: ELECTRICAL
*)
(*@KEY@:DESCRIPTION*)
version 1.0	13. nov. 2008
programmer 	oscat
tested by	hugo

click_mode decodes an input for single, double or long click and sets the corresponding output single, doulbe or long.
the input configures itself to be high or low active depending on which state the input stays longer than t_reconfig.
(*@KEY@:END_DESCRIPTION*)
FUNCTION_BLOCK CLICK_MODE

(*Group:Default*)

VAR_INPUT
	IN :	BOOL;
	T_LONG :	TIME := T#500ms;
END_VAR

VAR_OUTPUT
	SINGLE :	BOOL;
	DOUBLE :	BOOL;
	LONG :	BOOL;
	TP_LONG :	BOOL;
END_VAR

VAR
	Timer :	TP;
	cnt :	INT;
	last :	BOOL;
END_VAR

(*@KEY@: WORKSHEET
NAME: CLICK_MODE
IEC_LANGUAGE: ST
*)
(* when input goes high start the timer to decode pulses *)
timer(in := IN, PT := T_LONG);
single := FALSE;
double := FALSE;

IF timer.Q THEN
	(* decode pulses while the timer is active *)
	IF NOT in AND last THEN	cnt := cnt + 1; END_IF;
ELSE
	CASE cnt OF
		1 : single := TRUE;
		2 : double := TRUE;
	END_CASE;
	cnt := 0;
END_IF;
last := in;
TP_LONG := NOT timer.Q AND (NOT LONG) AND IN;
LONG := NOT timer.Q AND in;

(* revision history

hm	13. nov. 2008	rev 1.0
	original release

*)
(*@KEY@: END_WORKSHEET *)
END_FUNCTION_BLOCK

(* ---- DEBOUNCE.ST ---- *)
(*@PROPERTIES_EX@
TYPE: POU
LOCALE: 0
IEC_LANGUAGE: ST
PLC_TYPE: independent
PROC_TYPE: independent
GROUP: ELECTRICAL
*)
(*@KEY@:DESCRIPTION*)
version 1.0	22. sep. 2008
programmer 	oscat
tested by	tobias

DEBOUNCE is used to debounce switch inputs.
in addition to the debounce functionality this FB can also be used to detect rising edges on IN when PM = TRUE.
When PM = FALSE, Q follows in with the debounce functionality.
(*@KEY@:END_DESCRIPTION*)
FUNCTION_BLOCK DEBOUNCE

(*Group:Default*)

VAR_INPUT
	IN :	BOOL;
	TD :	TIME;
	PM :	BOOL;
END_VAR

VAR_OUTPUT
	Q :	BOOL;
END_VAR

VAR
	deb :	TOF;
END_VAR

(*@KEY@: WORKSHEET
NAME: DEBOUNCE
IEC_LANGUAGE: ST
*)
IF NOT deb.Q AND IN THEN
	(* rising edge on input detetced and debounce timer elapsed *)
	Q := TRUE;
ELSIF NOT PM THEN
	Q := deb.Q;
ELSE
	Q := FALSE;
END_IF;

(* run debounce timer *)
deb(IN := IN, PT := TD);

(*
hm 22. sep. 2008	rev 1.0
	original version

*)
(*@KEY@: END_WORKSHEET *)
END_FUNCTION_BLOCK

(* ---- DIMM_2.ST ---- *)
(*@PROPERTIES_EX@
TYPE: POU
LOCALE: 0
IEC_LANGUAGE: ST
PLC_TYPE: independent
PROC_TYPE: independent
GROUP: ELECTRICAL
*)
(*@KEY@:DESCRIPTION*)
version 1.0	22. mar. 2009
programmer 	hugo
tested by	tobias

this is an intelligent dimmer interface with an autoset feature using double switch inputs
a configurable debounce timer will debounce the input signals
if t_on_max is set to anything other then 0 the output will be turned off after the max on time is reached.
the times for debounce, dimming ramp, wait time before dimming and max on time are all programmable.

the dimmer has outputs Q for on and off and also out with the analog dimm value.
two additional outputs d1 and d2 decode double clicks on i1 and i2.
(*@KEY@:END_DESCRIPTION*)
FUNCTION_BLOCK DIMM_2

(*Group:Default*)

VAR_INPUT
	SET :	BOOL;
	VAL :	BYTE := BYTE#255;
	I1 :	BOOL;
	I2 :	BOOL;
	RST :	BOOL;
	T_DEBOUNCE :	TIME := T#10ms;
	T_ON_MAX :	TIME := T#0h;
	T_DIMM_START :	TIME := T#1s;
	T_DIMM :	TIME := T#3s;
	MIN_ON :	BYTE := BYTE#50;
	MAX_ON :	BYTE := BYTE#255;
	RST_OUT :	BOOL;
	SOFT_DIMM :	BOOL := TRUE;
	DBL1_TOG :	BOOL;
	DBL2_TOG :	BOOL;
	DBL1_SET :	BOOL;
	DBL2_SET :	BOOL;
	DBL1_POS :	BYTE;
	DBL2_POS :	BYTE;
END_VAR

VAR_OUTPUT
	Q :	BOOL;
	D1 :	BOOL;
	D2 :	BOOL;
END_VAR

VAR_IN_OUT
	OUT :	BYTE := BYTE#0;
END_VAR

VAR
	t1 :	TOF;
	t2 :	TOF;
	dc1 :	CLICK_MODE;
	dc2 :	CLICK_MODE;
	t3 :	TON;
	dim :	_RMP_B;
END_VAR

(*@KEY@: WORKSHEET
NAME: DIMM_2
IEC_LANGUAGE: ST
*)
(* debouncing for inputs i1 and i2 *)
t1(IN := I1, PT := T_DEBOUNCE);
t2(IN := I2, PT := T_DEBOUNCE);
dc1(in := t1.Q, T_LONG := T_DIMM_START);
dc2(in := t2.Q, T_LONG := T_DIMM_START);

IF RST THEN
	IF RST_OUT THEN out := BYTE#0; END_IF;
	Q := FALSE;
	D1 := FALSE;
	D2 := FALSE;
ELSIF set THEN
	OUT := VAL;
	Q := TRUE;
ELSIF dc1.SINGLE THEN
	(* single click on i1 turns the dimmer on *)
	out := LIMIT(MAX(MIN_ON,BYTE#1), out, MAX_ON);
	Q := TRUE;
ELSIF dc2.SINGLE THEN
	(* single click on i2 turns the dimmer off *)
	Q := FALSE;
ELSIF dc1.TP_LONG THEN
	(* continuous on at i1 dimms up *)
	IF NOT Q THEN
		out := SEL(SOFT_DIMM, LIMIT(MAX(MIN_ON,BYTE#1), out, MAX_ON), BYTE#1);
	END_IF;
	Q := TRUE;
	dim.DIR := TRUE;
ELSIF dc2.TP_LONG THEN
	(* continuous on at i2 dimms down *)
	dim.DIR := FALSE;
END_IF;

(* set the double click output *)
IF NOT DBL1_TOG THEN D1 := FALSE; END_IF;
IF dc1.DOUBLE THEN
	IF DBL1_SET THEN
		OUT := DBL1_POS;
		Q := TRUE;
	ELSE
		D1 := NOT D1;
	END_IF;
END_IF;
IF NOT DBL2_TOG THEN D2 := FALSE; END_IF;
IF dc2.DOUBLE THEN
	IF DBL2_SET THEN
		OUT := DBL2_POS;
		Q := TRUE;
	ELSE
		D2 := NOT D2;
	END_IF;
END_IF;

(* while dimming is active ramp the output out up or down *)
dim(dir := dc2.LONG, e := dc1.LONG OR dc2.LONG , TR := T_DIMM, rmp := out);
out := dim.RMP;

(* turn off output if a value of 0 is reached *)
IF out = BYTE#0 THEN Q := FALSE; END_IF;

(* limit the maximum runtime *)
IF t_ON_MAX > t#0s THEN
	t3(in := q, pt := T_ON_MAX);
	Q := Q XOR t3.Q;
END_IF;

(* revision history

hm 22. mar. 2009	rev 1.0
	original version

*)
(*@KEY@: END_WORKSHEET *)
END_FUNCTION_BLOCK

(* ---- DIMM_I.ST ---- *)
(*@PROPERTIES_EX@
TYPE: POU
LOCALE: 0
IEC_LANGUAGE: ST
PLC_TYPE: independent
PROC_TYPE: independent
GROUP: ELECTRICAL
*)
(*@KEY@:DESCRIPTION*)
version 2.3	26. jan. 2009
programmer 	hugo
tested by	tobias

this is an intelligent dimmer interface with an autoset feature for "in" it will automatically detect the type of switch:
low active pulses or high high active pulses are allowd for in.
a configurable debounce timer will debounce input signals
if t_on_max is set to anything other then 0 the output will be turned off after the max on time is reached.
the times for debounce, dimming ramp, wait time before dimming and max on time are all programmable.

the dimmer has outputs Q for on and off and also out with the analog dimm value.
(*@KEY@:END_DESCRIPTION*)
FUNCTION_BLOCK DIMM_I

(*Group:Default*)

VAR_INPUT
	SET :	BOOL;
	VAL :	BYTE := BYTE#255;
	IN :	BOOL;
	RST :	BOOL;
	T_DEBOUNCE :	TIME := T#10ms;
	T_RECONFIG :	TIME := T#10s;
	T_ON_MAX :	TIME := T#0h;
	T_DIMM_START :	TIME := T#1s;
	T_DIMM :	TIME := T#3s;
	MIN_ON :	BYTE := BYTE#50;
	MAX_ON :	BYTE := BYTE#255;
	SOFT_DIMM :	BOOL := TRUE;
	DBL_TOGGLE :	BOOL;
	RST_OUT :	BOOL;
END_VAR

VAR_OUTPUT
	Q :	BOOL;
	DBL :	BOOL;
END_VAR

VAR_IN_OUT
	OUT :	BYTE := BYTE#0;
END_VAR

VAR
	config :	SW_RECONFIG;
	decode :	CLICK_MODE;
	t3 :	TON;
	dim :	_RMP_B;
	dir :	BOOL;
END_VAR

(*@KEY@: WORKSHEET
NAME: DIMM_I
IEC_LANGUAGE: ST
*)
(* the input is first sent through auto reconfiguration and debouncing *)
config(IN := IN, TD := T_DEBOUNCE, TR := T_RECONFIG);
decode(in := config.Q, T_LONG := T_DIMM_START);

IF RST THEN
	IF rst_out THEN out := BYTE#0; END_IF;
	Q := FALSE;
	dir := out > BYTE#127;
ELSIF set THEN
	out := val;
	Q := TRUE;
	(* set direction to up when value < 127 otherwise set dir down dir is reversed because next action will reverse again *)
	dir := out > BYTE#127;
ELSIF decode.SINGLE THEN
	(* a single click reverses output Q *)
	Q := NOT Q;
	(* when dimmer is turned on we need to limit out to min and max limits *)
	IF Q THEN OUT := INT_TO_BYTE(LIMIT_INT(MAX(_BYTE_TO_INT(MIN_ON),1), _BYTE_TO_INT(out), _BYTE_TO_INT(MAX_ON)));	END_IF;
	(* set the appropriate direction of dimmer dir is reversed because next action will reverse again *)
	dir := OUT > BYTE#127;
ELSIF decode.TP_LONG THEN
	IF NOT Q THEN
		IF SOFT_DIMM THEN
			OUT := BYTE#1;
			dir := TRUE;
		ELSE
            out := INT_TO_BYTE(LIMIT_INT(MAX(_BYTE_TO_INT(MIN_ON),1), _BYTE_TO_INT(out), _BYTE_TO_INT(MAX_ON)));
			DIR := out < BYTE#127;
		END_IF;
		Q := TRUE;
	ELSE
		(* reverse direction with every long click *)
		dir := NOT dir;
	END_IF;
END_IF;

(* set the double click output *)
IF NOT dbl_toggle THEN dbl := FALSE; END_IF;
IF decode.DOUBLE THEN dbl := NOT dbl; END_IF;

(* while dimming is active ramp the output out up or down *)
dim(DIR := dir, e := decode.LONG AND Q, TR := T_DIMM, rmp := out);
OUT := dim.RMP;
(* reverse direction when limits are reached *)
IF out = BYTE#0 THEN
	dir := TRUE;
ELSIF out = BYTE#255 THEN
	dir := FALSE;
END_IF;

(* limit the maximum runtime *)
IF t_ON_MAX > t#0s THEN
	t3(in := q, pt := T_ON_MAX);
	Q := Q XOR t3.Q;
END_IF;

(* revision history

hm 22.1.2007		rev 1.1
	deleted unused structure ramp

hm 2.feb 2007		rev 1.2
	changed structure to read time() at the beginning for better time consistency if a higher priorized tak interrupts dimm_i
	added statements in case structure for state 1 to allow for short 1 cycle input pulses

hm 	15.9.2007		rev 1.3
	replaced Time() with T_PLC_MS for compatibility and performance reasons

hm	30. sep. 2008	rev 1.4
	added Input VAL to supply value for set input
	added setup parameter init_val

hm	22. oct. 2008	rev 2.0
	new code and features

hm	14. nov. 2008	rev 2.1
	added soft_dimm feature

hm	16. nov. 2008	rev 2.2
	added reset out feature

hm	26. jan. 2009	rev 2.3
	dimming will also reverse at out = 0
	rst will override set
*)
(*@KEY@: END_WORKSHEET *)
END_FUNCTION_BLOCK

(* ---- F_LAMP.ST ---- *)
(*@PROPERTIES_EX@
TYPE: POU
LOCALE: 0
IEC_LANGUAGE: ST
PLC_TYPE: independent
PROC_TYPE: independent
GROUP: ELECTRICAL
*)
(*@KEY@:DESCRIPTION*)
version 1.2	22. oct. 2008
programmer 	hugo
tested by	oscat

F_Lamp is an interface to flourescent lamps. its main purpose is to protect flourescent lamps from dimming within the first T_NO_DIMM Time.
If Flourescent Lamps are dimmed during the first 100 hours the lifetime of the lamp is reduced dramatically.
The interface also counts ontime and cycles of the lamp for maintanance purposes.
(*@KEY@:END_DESCRIPTION*)
FUNCTION_BLOCK F_LAMP

(*Group:Default*)

VAR_INPUT
	SWITCH :	BOOL;
	DIMM :	BYTE := BYTE#255;
	RST :	BOOL;
	T_NO_DIMM :	UINT := UINT#100;
	T_MAINTENANCE :	UINT := UINT#15000;
END_VAR

VAR_OUTPUT
	LAMP :	BYTE;
	STATUS :	BYTE;
END_VAR

VAR_IN_OUT
	ONTIME :	UDINT;
	CYCLES :	UDINT;
END_VAR

VAR
	runtime :	ONTIME;
END_VAR

(*@KEY@: WORKSHEET
NAME: F_LAMP
IEC_LANGUAGE: ST
*)
runtime(in := switch, SECONDS := ONTIME , CYCLES := CYCLES);
CYCLES := runtime.CYCLES;
ONTIME := runtime.SECONDS;

IF RST THEN
	ONTIME := UDINT#0;
	CYCLES := UDINT#0;
END_IF;
IF SWITCH THEN
	IF ontime < UINT_TO_UDINT(T_NO_DIMM) * UDINT#3600 THEN
		LAMP := BYTE#255;
		STATUS := BYTE#111;
	ELSE
		LAMP := DIMM;
		STATUS := BYTE#112;
	END_IF;
ELSE
	LAMP := BYTE#0;
	STATUS := BYTE#110;
END_IF;

IF ontime >= UINT_TO_UDINT(T_maintenance) * UDINT#3600 AND T_Maintenance > UINT#0 THEN
	STATUS := BYTE#120;
END_IF;

(* revision history
hm	8. feb. 2007	rev 1.1
	original version

hm	22. oct. 2008	rev 1.2
	changed use of ontime for ontime 2.0
	ontime is now in seconds not hours
*)
(*@KEY@: END_WORKSHEET *)
END_FUNCTION_BLOCK

(* ---- HEAT_METER.ST ---- *)
(*@PROPERTIES_EX@
TYPE: POU
LOCALE: 0
IEC_LANGUAGE: ST
PLC_TYPE: independent
PROC_TYPE: independent
GROUP: HLK
*)
(*@KEY@:DESCRIPTION*)
version 1.10	23. jan. 2011
programmer 		hugo
tested by		oscat

Heat meter measures the heat transfer of water of a mixture of water and another component.
The inputs are foreward temperature and reverse temperature.
the additional component is specified with its parameters density, Specific heat capacity and content in %.
an input e anables the measurement while it can be configured to be based on X liters / pulse or in liters / hour.
the output Y is in Joule.
(*@KEY@:END_DESCRIPTION*)
FUNCTION_BLOCK HEAT_METER

(*Group:Default*)

VAR_INPUT
	TF :	REAL;
	TR :	REAL;
	LPH :	REAL;
	E :	BOOL;
	RST :	BOOL;
	CP :	REAL;
	DENSITY :	REAL;
	CONTENT :	REAL;
	PULSE_MODE :	BOOL;
	RETURN_METER :	BOOL;
	AVG_TIME :	TIME := T#5s;
END_VAR

VAR_OUTPUT
	C :	REAL;
END_VAR

VAR_IN_OUT
	Y :	REAL;
END_VAR

VAR
	tx :	UDINT;
	last :	UDINT;
	int1 :	FT_INT2;
	edge :	BOOL;
	x :	REAL;
	init :	BOOL;
	Y_last :	REAL;
	T_PLC_MS :	T_PLC_MS;
	WATER_ENTHALPY :	WATER_ENTHALPY;
	wa_TF :	REAL;
	wa_TR :	REAL;
END_VAR

(*@KEY@: WORKSHEET
NAME: HEAT_METER
IEC_LANGUAGE: ST
*)
IF rst THEN
	int1(rst := TRUE);
	int1.rst := FALSE;
	C := 0.0;
	Y := 0.0;
ELSIF e THEN
	water_enthalpy(T:=TF);
	wa_TF:=water_enthalpy.Result;

	water_enthalpy(T:=TR);
	wa_TR:=water_enthalpy.Result;

	X := (WATER_DENSITY(SEL(return_meter, TF, TR), FALSE) * (wa_TF - wa_TR) * (1.0 - content) + CP * Density * content * (TF-TR));
END_IF;

(* integrate or add consumption *)
int1(run := NOT pulse_mode AND e, in := X * LPH * 2.77777777777E-4);
IF pulse_mode THEN
	IF NOT edge AND E THEN Y := Y + X * LPH; END_IF;
ELSE
	Y := int1.Out;
END_IF;

(* store the value of e *)
edge := e;

(* read system_time *)
T_PLC_MS();
tx:= T_PLC_MS.T_PLC_MS;

(* only init at startup necessary *)
IF NOT init THEN
	init := TRUE;
	last := tx;
END_IF;

(* calculate the current consumption *)
IF (tx - last >= TIME_TO_UDINT(AVG_TIME)) AND (avg_time > T#0s) THEN
	last := tx;
	C := (Y - Y_last) * 3.6E12 / TIME_TO_REAL(AVG_TIME);
	Y_last := Y;
END_IF;

(* revision history
hm	16. nov. 2007	rev 1.0
	original version

hm	24. dec. 2007	rev 1.1
	added config variable return_meter
	added output C for current consumption

hm	6. mar. 2008	rev 1.2
	corrected an error in pulse mode

hm	16. mar. 2008	rev 1.3
	added type conversion to avoid warnings under codesys 3.0

hm	21. oct. 2008	rev 1.4
	improved code

hm	6. nov. 2008	rev 1.5
	changed to FT_INT2 to avoid overrun at hig values

hm	8. feb. 2009	rev 1.6
	changes Y to be I/O

hm	23. mar. 2009	rev 1.7
	real constants updated to new systax using dot
	corected error in formula

hm	27. jul 2009	rev 1.8
	output C is now calculated in J/h

hm	13. nov. 2009	rev 1.9
	output C is now calculated correctly

hm	23. jan. 2011	rev 1.10
	corrected an error with pulse_mode
*)
(*@KEY@: END_WORKSHEET *)
END_FUNCTION_BLOCK

(* ---- HEAT_TEMP.ST ---- *)
(*@PROPERTIES_EX@
TYPE: POU
LOCALE: 0
IEC_LANGUAGE: ST
PLC_TYPE: independent
PROC_TYPE: independent
GROUP: HLK
*)
(*@KEY@:DESCRIPTION*)
version 1.2	13. mar. 2009
programmer 	hugo
tested by	oscat

Heat_Temp calculates a heat characteristic based on the formula: tv=ti+(tvmax-ti)*((ti-tau)/(ti-taumin))^(1/n)
while
tv necessary heating temperature.
ti internal room temperature (20°C)
tau current external temperature
taumin external temperature to determine characteristics
C exponent for heating system (normally 1,33 or 1,1 for floor heating)

The two additional inputs TY_min and TY_max set limits for the output TY, while an offset inputs allows to rise or lower the room temperature.
(*@KEY@:END_DESCRIPTION*)
FUNCTION_BLOCK HEAT_TEMP

(*Group:Default*)

VAR_INPUT
	T_EXT :	REAL;
	T_INT :	REAL;
	OFFSET :	REAL;
	T_REQ :	REAL;
	TY_MAX :	REAL := REAL#70.0;
	TY_MIN :	REAL := REAL#25.0;
	TY_CONFIG :	REAL := REAL#70.0;
	T_INT_CONFIG :	REAL := REAL#20.0;
	T_EXT_CONFIG :	REAL := REAL#-15.0;
	T_DIFF :	REAL := REAL#10.0;
	C :	REAL := REAL#1.33;
	H :	REAL := REAL#3.0;
END_VAR

VAR_OUTPUT
	TY :	REAL;
	HEAT :	BOOL;
END_VAR

VAR
	tr :	REAL;
	tx :	REAL;
END_VAR

(*@KEY@: WORKSHEET
NAME: HEAT_TEMP
IEC_LANGUAGE: ST
*)
tr := T_INT + OFFSET;
tx := (tr - T_EXT) / (T_INT_CONFIG - T_EXT_CONFIG);

IF T_EXT + H > tr THEN
	TY := 0.0;
ELSE
	TY := LIMIT(TY_MIN, tr + T_DIFF * 0.5 * tx + (TY_CONFIG - T_DIFF * 0.5 - tr) * EXPT(tx, 1.0 / C), TY_MAX);
END_IF;

TY := MAX(TY, T_REQ);
HEAT := TY > 0.0;

(*

tv=ti+(tvmax-ti)*((ti-tau)/(ti-taumin))^(1/n)

tv aktuelle Vorlauftemp.
ti Raumtemperatur innen (20°C)
tau aktuelle Außentemperatur
taumin minimale Außentemperatur -12°C oder -15°C
n Heizkörperexponent (meistens 1,33)
Fußbodenheizung = 1,1
Wandheizung 1,3

Normen z. B. DIN 4703, DIN 4725 oder die Literatur, z. B Recknagel Abschnitt 1.3.5.

*)

(* revision history
hm	27. jan. 2008	rev 1.0
	original version

hm	26. sep. 2008	rev 1.1
	moved T_INT from config to Input
	added config variable H
	corrected error in formula

hm	13. mar. 2009	rev 1.2
	improved code

*)
(*@KEY@: END_WORKSHEET *)
END_FUNCTION_BLOCK

(* ---- LEGIONELLA.ST ---- *)
(*@PROPERTIES_EX@
TYPE: POU
LOCALE: 0
IEC_LANGUAGE: ST
PLC_TYPE: independent
PROC_TYPE: independent
GROUP: HLK
*)
(*@KEY@:DESCRIPTION*)
version 1.3	13. mar. 2009
programmer 	oscat
tested by	oscat

Legionella is a complete sequencer for up to 8 hot water lines that need to be sterilzed periodically.
legionella needs a DT input with the appropriate time, usually gererated by the rtc of the system. for system independence this time is connected externally.
T_start is the time when sterilazation should be started and day is the day_of_week when it should be performed (1=Monday and 7=sunday).
so sterilazation is autioimatically performed once a week at a specified time.
temp_set and temp_hys and temp_offset specify the boiler temperatur nedded for sterilization. as a defaut Temp_set is set to 70 deg C and Temp_hys is set to 5 deg C and temp_offset is 10 deg C.
a temp boiler input reads the boiler temperature of the hot water tank.
after a start pulse is gererated by the weekly timer or a manual test input the sequence is started:
1. the boiler is heated to temp_set + temp_offset + temp_hys = 85 deg C unless chaged at setup.
	the heat output is turned on and tells the heater to turn heating on. if the temp is not reached for a time of t_max_heat (10 min) the error output is set and the sequence is stopped.
2. after the specified temperature is reached, the output valve0 and pump is turned on and starts sterilization of line0 until temp_return has reached temp_set and continues to sterilize for a time of tp_0 (5 min default).
	if tmep_set is not reached at the temp_return_input then the error output is set and the sequence will be stopped.
	if there is no temp sensor for temp_return (the temperature at the return point for the circulation pump pls set this imput to a value greater then temp_set (by default use 100 deg C).
	in this case sterilization is performed for the default times without monitoring the return temp.
3. this sequence is repeated for up to valves.

connection scheme:

temp_boiler:	input oif the boiler temperature sensor.
temp_hys:		config value for the heater hysteresis, preset to 5 deg C.
temp_offset:	config value for the heater temp_offset against temp_set, preset to 10 deg C.
temp_set:		config value for the specified sterilization temperature, preset to 70 deg C.
temp_return:	input of the circulation return line temperature sensor, if not availabe set this value to 100 deg C.
manual:		manual input to start the sterilization by hand for diagnostic purposes, rising edge active, leave low for automatic operation.
DT_in:			date,time input supplied by a external real time clock.
T_start:		time of day when the sterilization should be started.
day:			config value for day of week when the process should be started, preset to sunday.
t_max_hest:	tmax time to be needed for the heater to heat the hot water tank to the specified value, preset to 10 min.
(*@KEY@:END_DESCRIPTION*)
FUNCTION_BLOCK LEGIONELLA

(*Group:Default*)

VAR_INPUT
	MANUAL :	BOOL;
	TEMP_BOILER :	REAL;
	TEMP_RETURN :	REAL := 100.0;
	DT_IN :	UDINT;
	RST :	BOOL;
	T_START :	UDINT := UDINT#10800000;(*tod#03:00:00*)
	DAY :	INT := 7;
	TEMP_SET :	REAL := 70.0;
	TEMP_OFFSET :	REAL := 10.0;
	TEMP_HYS :	REAL := 5.0;
	T_MAX_HEAT :	TIME := t#10m;
	T_MAX_RET :	TIME := t#10m;
	TP_0 :	TIME := t#5m;
	TP_1 :	TIME := t#5m;
	TP_2 :	TIME := t#5m;
	TP_3 :	TIME := t#5m;
	TP_4 :	TIME := t#5m;
	TP_5 :	TIME := t#5m;
	TP_6 :	TIME := t#5m;
	TP_7 :	TIME := t#5m;
END_VAR

VAR_OUTPUT
	HEAT :	BOOL;
	PUMP :	BOOL;
	VALVE0 :	BOOL;
	VALVE1 :	BOOL;
	VALVE2 :	BOOL;
	VALVE3 :	BOOL;
	VALVE4 :	BOOL;
	VALVE5 :	BOOL;
	VALVE6 :	BOOL;
	VALVE7 :	BOOL;
	RUN :	BOOL;
	STATUS :	BYTE;
END_VAR

VAR
	X1 :	timer_1;
	x2 :	sequence_8;
	x3 :	hyst_1;
	init :	BOOL;
END_VAR

(*@KEY@: WORKSHEET
NAME: LEGIONELLA
IEC_LANGUAGE: ST
*)
(* startup initialization *)
IF NOT init THEN
	init := TRUE;
	X1.day := SHR(BYTE#128,day);
	X1.start := T_start;
	X3.low := Temp_offset + temp_set;
	X3.high := Temp_hys + X3.low;
	X2.wait0 := T_max_heat;
	X2.delay0 := TP_0;
	X2.delay1 := TP_1;
	X2.delay2 := TP_2;
	X2.delay3 := TP_3;
	X2.delay4 := TP_4;
	X2.delay5 := TP_5;
	X2.delay6 := TP_6;
	X2.delay7 := TP_7;
	X2.wait1 := T_max_ret;
	X2.wait2 := T_max_ret;
	X2.wait3 := T_max_ret;
	X2.wait4 := T_max_ret;
	X2.wait5 := T_max_ret;
	X2.wait6 := T_max_ret;
	X2.wait7 := T_max_ret;
	X2();
END_IF;

(* oerational code *)
X1(DTi := DT_in);
IF X1.Q OR MANUAL OR x2.run THEN
	X3(in := temp_boiler);
	X2.in0 := X3.Q OR x3.win;
	X2.in1 := temp_return >= temp_set;
	X2.in2 := x2.in1;
	X2.in3 := x2.in1;
	X2.in4 := x2.in1;
	X2.in5 := x2.in1;
	X2.in6 := x2.in1;
	X2.in7 := x2.in1;
	X2.rst := rst;
	X2(start := X1.Q OR MANUAL);
	run := x2.run;
	pump := x2.QX;
	Heat := NOT X3.Q AND x2.run;
	valve0 := X2.Q0;
	valve1 := X2.Q1;
	valve2 := X2.Q2;
	valve3 := X2.Q3;
	valve4 := X2.Q4;
	valve5 := X2.Q5;
	valve6 := X2.Q6;
	valve7 := X2.Q7;
	pump := X2.QX;
	status := X2.status;
ELSE;
	X2(start := FALSE);
	status := x2.status;
END_IF;

(* revision history

hm 17.jan 2007	rev 1.1
	rewritten to st for higher performance
	changes eeror output to esr compatible status output

hm	23. 10.2008	rev 1.2
	update code to use new version of timer_1

hm	13. mar. 2009	rev 1.3
	real constants updated to new systax using dot

*)
(*@KEY@: END_WORKSHEET *)
END_FUNCTION_BLOCK

(* ---- PULSE_LENGTH.ST ---- *)
(*@PROPERTIES_EX@
TYPE: POU
LOCALE: 0
IEC_LANGUAGE: ST
PLC_TYPE: independent
PROC_TYPE: independent
GROUP: ELECTRICAL
*)
(*@KEY@:DESCRIPTION*)
version 1.1	15 sep 2007
programmer 	oscat
tested by		tobias

Pulse_length indicates on 3 outputs if an input pulse had been shorter than T_short (short = True), longer than T_long (long = True) or between T_short and T_long (middle = True).
(*@KEY@:END_DESCRIPTION*)
FUNCTION_BLOCK PULSE_LENGTH

(*Group:Default*)

VAR_INPUT
	IN :	BOOL;
	T_SHORT :	TIME := T#100ms;
	T_LONG :	TIME := T#1s;
END_VAR

VAR_OUTPUT
	SHORT :	BOOL;
	MIDDLE :	BOOL;
	LONG :	BOOL;
END_VAR

VAR
	tx :	TIME;
	tn :	TIME;
	edge :	BOOL;
	T_PLC_MS :	T_PLC_MS;
END_VAR

(*@KEY@: WORKSHEET
NAME: PULSE_LENGTH
IEC_LANGUAGE: ST
*)
(* read system time *)

T_PLC_MS();
tx:= UDINT_TO_TIME(T_PLC_MS.T_PLC_MS);

(* reset outputs, they should only be active 1 cycle *)
short := FALSE;
Middle := FALSE;
long := FALSE;

(* detect rising edge *)
IF in AND NOT edge THEN
	edge := TRUE;
	tn := tx;

(* detect for falling edge *)
ELSIF NOT in AND edge THEN
	edge := FALSE;
	tn := tx - tn;
	IF tn < t_short THEN
		short := TRUE;
	ELSIF tn > t_long THEN
		long := TRUE;
	ELSE
		Middle := TRUE;
	END_IF;

(* generate long pulse as soon as T_long is reached *)
ELSIF in AND tx - tn > t_long THEN
	long := TRUE;
END_IF;

(* revision history

hm	15. feb 2006	rev 1.0
	original version

hm	15 sep 2007		rev 1.1
	replaced Time() with T_PLC_MS for compatibility and performance reasons

*)
(*@KEY@: END_WORKSHEET *)
END_FUNCTION_BLOCK

(* ---- PULSE_T.ST ---- *)
(*@PROPERTIES_EX@
TYPE: POU
LOCALE: 0
IEC_LANGUAGE: ST
PLC_TYPE: independent
PROC_TYPE: independent
GROUP: ELECTRICAL
*)
(*@KEY@:DESCRIPTION*)
version 1.0	15. jul. 2008
programmer 	hugo
tested by	oscat

PULSE_T generates a pulse of length T2 if the input pulse is shorter than T1.
if the input pulse is longer than T1, the output follows the input.
and rising edge on in will kill a possible output pulse and generate a new pulse instead.
(*@KEY@:END_DESCRIPTION*)
FUNCTION_BLOCK PULSE_T

(*Group:Default*)

VAR_INPUT
	IN :	BOOL;
	T1 :	TIME;
	T2 :	TIME;
	RST :	BOOL;
END_VAR

VAR_OUTPUT
	Q :	BOOL;
END_VAR

VAR
	init :	BOOL;
	last :	TIME;
	tx :	TIME;
	edge :	BOOL;
	T_PLC_MS :	T_PLC_MS;
END_VAR

(*@KEY@: WORKSHEET
NAME: PULSE_T
IEC_LANGUAGE: ST
*)
(* read system time *)
T_PLC_MS();
tx:= UDINT_TO_TIME(T_PLC_MS.T_PLC_MS);

IF NOT init THEN
	init := TRUE;
	last := tx;
ELSIF RST THEN
	(* asynchronous reset *)
	Q := FALSE;
ELSIF IN AND NOT edge AND NOT Q THEN
	(* a rising edge on in will reversre the output status, if new pulse is startet the start time is stored in last *)
	last := tx;
	Q := TRUE;
ELSIF NOT IN AND edge AND ((tx - last) > T1) THEN
	(* a falling edge on IN will clear the output if in was high for more then T1 *)
	Q := FALSE;
ELSIF (tx - last) >= T2 THEN
	(* timeout for long pulse if second click did not occur or in stays high *)
	Q := FALSE;
END_IF;

edge := IN;

(* revision histroy
hm	15. jul. 2008	rev 1.0
	original release

*)
(*@KEY@: END_WORKSHEET *)
END_FUNCTION_BLOCK

(* ---- SW_RECONFIG.ST ---- *)
(*@PROPERTIES_EX@
TYPE: POU
LOCALE: 0
IEC_LANGUAGE: ST
PLC_TYPE: independent
PROC_TYPE: independent
GROUP: ELECTRICAL
*)
(*@KEY@:DESCRIPTION*)
version 1.0	22. oct. 2008
programmer 	hugo
tested by	oscat

SW_reconfig detects if an input is high or low active and debounces the input
(*@KEY@:END_DESCRIPTION*)
FUNCTION_BLOCK SW_RECONFIG

(*Group:Default*)

VAR_INPUT
	IN :	BOOL;
	TD :	TIME;
	TR :	TIME;
END_VAR

VAR_OUTPUT
	Q :	BOOL;
END_VAR

VAR
	T1 :	TON;
	T2 :	TON;
	INV :	BOOL;
END_VAR

(*@KEY@: WORKSHEET
NAME: SW_RECONFIG
IEC_LANGUAGE: ST
*)
(* run debounce circuit *)
t1(in := IN, PT := TD);

IF tr > t#0s THEN
	(* generate output *)
	Q := t1.Q XOR inv;
	(* reconfiguration timer *)
	T2(in := Q, pt := TR);
	(* when T2.Q goes high then reverse INV *)
	IF T2.Q THEN INV := NOT INV; END_IF;
ELSE
	Q := t1.Q;
END_IF;

(* revision history
hm	22.10.2008	rev 1.0
	original version

*)
(*@KEY@: END_WORKSHEET *)
END_FUNCTION_BLOCK

(* ---- SWITCH_I.ST ---- *)
(*@PROPERTIES_EX@
TYPE: POU
LOCALE: 0
IEC_LANGUAGE: ST
PLC_TYPE: independent
PROC_TYPE: independent
GROUP: ELECTRICAL
*)
(*@KEY@:DESCRIPTION*)
version 1.1	15 sep 2007
programmer 	oscat
tested by		tobias

this is an intelligent switch interface which has an autodetect feature for in and it will detect the type of switch connected automatically
the input can be connected to low active pulses, high active pulses and on/off switch.
it will automatically adjust to the correct type without manual adjustment
a configurable debounce timer will debounce input signals
if t_on_max is set to anything other then 0 the output will be turned off after the max on time is reached.
(*@KEY@:END_DESCRIPTION*)
FUNCTION_BLOCK SWITCH_I

(*Group:Default*)

VAR_INPUT
	SET :	BOOL;
	IN :	BOOL;
	RST :	BOOL;
	T_DEBOUNCE :	TIME := T#10ms;
	T_RECONFIG :	TIME := T#1s;
	T_ON_MAX :	TIME := T#0h;
END_VAR

VAR_OUTPUT
	Q :	BOOL := FALSE;
END_VAR

VAR
	state :	BYTE := BYTE#0;
	edge :	BOOL := FALSE;
	r_edge :	BOOL := FALSE;
	T_on :	TIME;
	tx :	TIME;
	T_PLC_MS :	T_PLC_MS;
END_VAR

(*@KEY@: WORKSHEET
NAME: SWITCH_I
IEC_LANGUAGE: ST
*)
(* read system time *)
T_PLC_MS();
tx:= UDINT_TO_TIME(T_PLC_MS.T_PLC_MS);

(* asynchronous set and reset first *)
IF set AND NOT rst THEN
	Q := TRUE;
	T_on := tx;
ELSIF rst THEN
	Q := FALSE;
(* check FOR input edge AND start debounce timer *)
ELSIF (in XOR edge) AND NOT (state = BYTE#1) THEN
	state := BYTE#1;
	T_on := Tx;
(* edge was detected and debounce time elapsed *)
ELSIF (state = BYTE#1) AND (Tx - t_debounce >= T_on) THEN
	state := BYTE#2;
	(* react on rising or falling edge depending on r_edge *)
	IF r_edge XOR in THEN Q := NOT Q; END_IF;
(* wait for T_reconfig and adjust r_edge *)
ELSIF state = BYTE#2 AND Tx - t_reconfig >= T_on THEN
	r_edge := in;
END_IF;
IF Q AND T_on_max > t#0ms AND Tx >= T_on + T_on_max THEN
	Q := FALSE;
END_IF;
edge := in;

(* revision history

hm	4 aug 2006	rev 1.0
	original version

hm	15.9.2007	rev 1.1
	replaced Time() with T_PLC_MS for compatibility and performance reasons

*)
(*@KEY@: END_WORKSHEET *)
END_FUNCTION_BLOCK

(* ---- SWITCH_X.ST ---- *)
(*@PROPERTIES_EX@
TYPE: POU
LOCALE: 0
IEC_LANGUAGE: ST
PLC_TYPE: independent
PROC_TYPE: independent
GROUP: ELECTRICAL
*)
(*@KEY@:DESCRIPTION*)
version 1.0	15 Feb 2007
programmer 	oscat
tested by	tobias
(*@KEY@:END_DESCRIPTION*)
FUNCTION_BLOCK SWITCH_X

(*Group:Default*)

VAR_INPUT
	IN1 :	BOOL;
	IN2 :	BOOL;
	IN3 :	BOOL;
	IN4 :	BOOL;
	IN5 :	BOOL;
	IN6 :	BOOL;
	T_DEBOUNCE :	TIME := T#50ms;
END_VAR

VAR_OUTPUT
	Q1 :	BOOL;
	Q2 :	BOOL;
	Q3 :	BOOL;
	Q4 :	BOOL;
	Q5 :	BOOL;
	Q6 :	BOOL;
	Q31 :	BOOL;
	Q41 :	BOOL;
	Q51 :	BOOL;
	Q61 :	BOOL;
	Q32 :	BOOL;
	Q42 :	BOOL;
	Q52 :	BOOL;
	Q62 :	BOOL;
END_VAR

VAR
	INIT :	BOOL;
	T1 :	TOF;
	T2 :	TOF;
	T3 :	TOF;
	T4 :	TOF;
	T5 :	TOF;
	T6 :	TOF;
	tx :	TIME;
	x1 :	BOOL;
	x2 :	BOOL;
	E1 :	BOOL;
	E2 :	BOOL;
END_VAR

(*@KEY@: WORKSHEET
NAME: SWITCH_X
IEC_LANGUAGE: ST
*)
(* initialize on startup *)
IF NOT init THEN
	init := TRUE;
	IF t_debounce < t#50ms THEN tx := t#50ms; ELSE tx := t_debounce; END_IF;
	T1(PT := Tx);
	T2(PT := Tx);
	T3(PT := Tx);
	T4(PT := Tx);
	T5(PT := Tx);
	T6(PT := Tx);
ELSE
	Q1 := FALSE;
	Q2 := FALSE;
	Q3 := FALSE;
	Q4 := FALSE;
	Q5 := FALSE;
	Q6 := FALSE;
	Q31 := FALSE;
	Q41 := FALSE;
	Q51 := FALSE;
	Q61 := FALSE;
	Q32 := FALSE;
	Q42 := FALSE;
	Q52 := FALSE;
	Q62 := FALSE;
END_IF;

(* read inputs and debounce *)
	T1(IN := IN1);
	T2(IN := IN2);
	T3(IN := IN3);
	T4(IN := IN4);
	T5(IN := IN5);
	T6(IN := IN6);

(* detect edge of IN1 and IN2 *)
IF t1.Q AND NOT E1 THEN X1 := TRUE; END_IF;
IF t2.Q AND NOT E2 THEN X2 := TRUE; END_IF;

IF t1.Q THEN
	IF t3.q THEN
		q31 := TRUE;
		X1 := FALSE;
	ELSIF t4.q THEN
		q41 := TRUE;
		X1 := FALSE;
	ELSIF t5.q THEN
		q51 := TRUE;
		X1 := FALSE;
	ELSIF t6.q THEN
		q61 := TRUE;
		X1 := FALSE;
	END_IF;
ELSIF t2.Q THEN
	IF t3.q THEN
		q32 := TRUE;
		X2 := FALSE;
	ELSIF t4.q THEN
		q42 := TRUE;
		X2 := FALSE;
	ELSIF t5.q THEN
		q52 := TRUE;
		X2 := FALSE;
	ELSIF t6.q THEN
		q62 := TRUE;
		X2 := FALSE;
	END_IF;
(* in1 was active alone *)
ELSIF NOT T1.Q AND E1 AND X1 THEN
	Q1 := TRUE;
	X1 := FALSE;
ELSIF NOT T2.Q AND E2 AND X2 THEN
	Q2 := TRUE;
	X2 := FALSE;
ELSIF T3.Q THEN
	Q3 := TRUE;
ELSIF T4.Q THEN
	Q4 := TRUE;
ELSIF T5.Q THEN
	Q5 := TRUE;
ELSIF T6.Q THEN
	Q6 := TRUE;
END_IF;

(* save state of in1 and in2 *)
E1 := T1.Q;
E2 := T2.Q;
(*@KEY@: END_WORKSHEET *)
END_FUNCTION_BLOCK

(* ---- T_AVG24.ST ---- *)
(*@PROPERTIES_EX@
TYPE: POU
LOCALE: 0
IEC_LANGUAGE: ST
PLC_TYPE: independent
PROC_TYPE: independent
GROUP: HLK
*)
(*@KEY@:DESCRIPTION*)
version 1.2	13. mar. 2009
programmer 	hugo
tested by	oscat

this function calculates the averaged daytime temperature by taking 48 samples over one day.
a trigger tp will be true for one cycle when the output is updated.
using the input scale the outputs can be adjusted to different scales.
(*@KEY@:END_DESCRIPTION*)
FUNCTION_BLOCK T_AVG24

(*Group:Default*)

VAR_INPUT
	TS :	INT;
	DTI :	UDINT;
	RST :	BOOL;
	T_FILTER :	TIME := T#10m;
	SCALE :	REAL := 1.0;
	OFS :	REAL;
END_VAR

VAR_OUTPUT
	TA :	REAL;
	TP :	BOOL;
END_VAR

VAR_IN_OUT
	T24 :	REAL;
	T24_MAX :	REAL;
	T24_MIN :	REAL;
END_VAR

VAR
	samples :	oscat_T_AVG24;
	pos :	INT;
	init :	BOOL;
	ft1 :	FILTER_I;
	sum :	DINT;
	last :	UDINT;
	tmp_max :	INT;
	tmp_min :	INT;
	i :	INT;
END_VAR

(*@KEY@: WORKSHEET
NAME: T_AVG24
IEC_LANGUAGE: ST
*)
(* first filter the sensor readings *)
ft1(X := TS, T := T_FILTER);

IF rst OR NOT init THEN
	init := TRUE;
	IF T24 = -1000.0 THEN t24 := INT_TO_REAL(ft1.Y) * 0.1; END_IF;
	FOR pos := 0 TO 47 DO
		samples[pos] := REAL_TO_INT(T24 * 10.0);
	END_FOR;
	pos := 0;
	sum := INT_TO_DINT(samples[0]) * DINT#48;
	(* calculate the output value *)
	TA := (INT_TO_REAL(ft1.Y) * 0.1 + OFS) * SCALE;
	T24 := (DINT_TO_REAL(sum) * 0.00208333333333 + OFS) * SCALE;
	tp := TRUE;
ELSIF (dti / UDINT#60 MOD UDINT#30) = UDINT#0 AND DTI > last THEN
	(* make sure we onlyexecute once every 30 mins *)
	last := DTI + TIME_TO_UDINT(T#1m);
	(* sample the temperature every 30 mins and store in ring buffer samples *)
	(* sum always holds the sum of the array *)
	(* subtract the oldest sample from sum *)
	sum := sum - INT_TO_DINT(samples[pos]);
	(* strore the new sample *)
	samples[pos] := ft1.Y;
	(* add the new sample to sum *)
	sum := sum + INT_TO_DINT(samples[pos]);
	(* increment the counter for the next sample *)
	pos := INC1(pos, 48);
	(* calculate the output value *)
	TA := (INT_TO_REAL(ft1.Y) * 0.1 + OFS) * SCALE;
	T24 := (DINT_TO_REAL(sum) * 0.00208333333333 + OFS) * SCALE;
	(* calculate the min and max over the last 24 hours *)
	tmp_max := -32000;
	tmp_min := 32000;
	FOR i := 0 TO 47 DO
		tmp_max := MAX(tmp_max, samples[i]);
		tmp_min := MIN(tmp_min, samples[i]);
	END_FOR;
	T24_MAX := (INT_TO_REAL(tmp_max) * 0.1 + OFS) * SCALE;
	T24_MIN := (INT_TO_REAL(tmp_min) * 0.1 + OFS) * SCALE;
	tp := TRUE;
ELSE
	tp := FALSE;
END_IF;

(* revision history
hm	3. nov. 2008	rev 1.0
	original version

hm	8. feb. 2009	rev 1.1
	changes sign of OFS
	added outputs t24_min and t24_max

hm	13. mar. 2009	rev 1.2
	improved code
*)
(*@KEY@: END_WORKSHEET *)
END_FUNCTION_BLOCK

(* ---- TANK_LEVEL.ST ---- *)
(*@PROPERTIES_EX@
TYPE: POU
LOCALE: 0
IEC_LANGUAGE: ST
PLC_TYPE: independent
PROC_TYPE: independent
GROUP: HLK
*)
(*@KEY@:DESCRIPTION*)
version 1.0	27 feb 2007
programmer 	hugo
tested by	tobias
(*@KEY@:END_DESCRIPTION*)
FUNCTION_BLOCK TANK_LEVEL

(*Group:Default*)

VAR_INPUT
	LEVEL :	BOOL;
	LEAK :	BOOL;
	ACLR :	BOOL;
	MAX_VALVE_TIME :	TIME;
	LEVEL_DELAY_TIME :	TIME;
END_VAR

VAR_OUTPUT
	VALVE :	BOOL;
	ALARM :	BOOL;
	STATUS :	BYTE;
END_VAR

VAR
	cx :	ACTUATOR_COIL;
	tn :	TON;
	tl :	TONOF;
	open :	BOOL;
END_VAR

(*@KEY@: WORKSHEET
NAME: TANK_LEVEL
IEC_LANGUAGE: ST
*)
(* preprocess the level information *)
tl(in := level, T_ON := level_delay_time, T_OFF := level_delay_time);
open := tl.Q;

(* start logic *)
IF ALARM THEN
	(* check for ACLR if ALARM is present *)
	IF ACLR THEN
		ALARM := FALSE;
		STATUS := BYTE#101; (* aclr pressed *)
		cx(in := FALSE);
	END_IF;
	RETURN;
ELSIF LEAK THEN
	(* leakeage detected *)
	cx(in := FALSE);
	ALARM := TRUE;
	STATUS := BYTE#1;	(* leakeage error *)
ELSIF open THEN
	(* valve needs to be opened because level is too low *)
	cx(in := TRUE);
	STATUS := BYTE#102; (* valve open by low level *)
ELSE
	(* valve needs to be closed *)
	cx(in := FALSE);
	STATUS := BYTE#100; (* valve idle *)
END_IF;

(* check if valve is open too long and generate alarm if necessary *)
tn(in := cx.out AND (MAX_VALVE_TIME > T#0s), PT := MAX_VALVE_TIME);
IF tn.Q THEN
	ALARM := TRUE;
	STATUS := BYTE#2; (* overtime error *)
	cx(in := FALSE);
END_IF;

(* set output signal *)
VALVE := cx.out;
(*@KEY@: END_WORKSHEET *)
END_FUNCTION_BLOCK
